KUKA KRL program: MyProgram_186().src

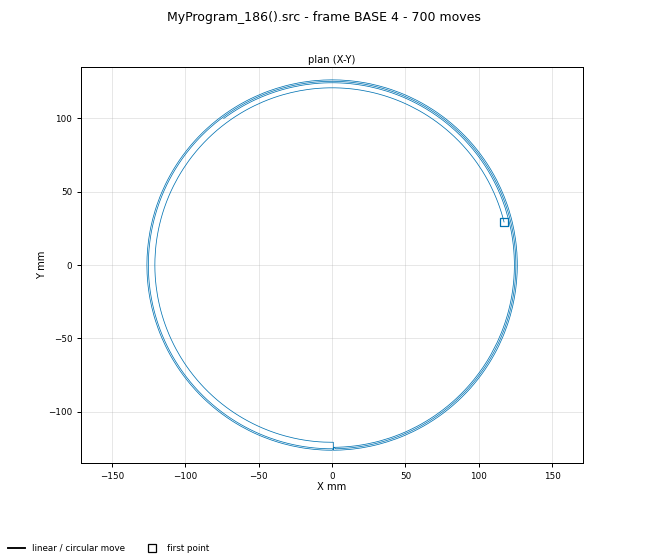
[picture p0: tool path of MyProgram_186().src in frame BASE 4, 700 of 700 moves have a stored position in this frame; points joined in program order, loops and branches not executed]
&ACCESS RVP
&REL 1
&PARAM TEMPLATE = C:\KRC\Roboter\Template\vorgabe
&PARAM EDITMASK = *
DEF MyProgram_186()
; ---- Setting reference (Base) ----
$BASE = BASE_DATA[4]

; --------------------------
; ---- Setting tool (TCP) ----
$TOOL = TOOL_DATA[3]
; --------------------------

$VEL.CP = VEL_APROX_PRINT
Startdeposition()
$VEL.CP = VEL_PRINT
LIN {X 117.2082,Y 29.362,Z 135,A 10.4187,B 24.9465,C -1.689,E1 25.1548,E2 795.6476} C_DIS
LIN {X 116.4539,Y 32.2231,Z 135,A 11.8113,B 24.9463,C -1.6929,E1 25.1537,E2 794.2539} C_DIS
LIN {X 115.5108,Y 35.4542,Z 135,A 13.5303,B 24.9456,C -1.7039,E1 25.1524,E2 792.5186} C_DIS
LIN {X 114.2566,Y 39.3095,Z 135,A 15.3056,B 24.9456,C -1.7024,E1 25.1508,E2 790.7568} C_DIS
LIN {X 113.2587,Y 42.0983,Z 135,A 16.7003,B 24.9454,C -1.7062,E1 25.1495,E2 789.3611} C_DIS
LIN {X 112.0398,Y 45.2414,Z 135,A 18.3803,B 24.9449,C -1.715,E1 25.1477,E2 787.6697} C_DIS
LIN {X 110.4582,Y 48.9779,Z 135,A 20.3068,B 24.9445,C -1.7207,E1 25.1456,E2 785.7402} C_DIS
LIN {X 109.0474,Y 52.0418,Z 135,A 21.6552,B 24.945,C -1.7129,E1 25.144,E2 784.4175} C_DIS
LIN {X 107.9261,Y 54.3318,Z 135,A 22.9862,B 24.9444,C -1.7224,E1 25.1423,E2 783.0713} C_DIS
LIN {X 106.3686,Y 57.3227,Z 135,A 24.664,B 24.9439,C -1.7307,E1 25.1401,E2 781.3826} C_DIS
LIN {X 104.398,Y 60.8384,Z 135,A 26.5827,B 24.9435,C -1.7363,E1 25.1375,E2 779.4606} C_DIS
LIN {X 102.3123,Y 64.2836,Z 135,A 28.5381,B 24.943,C -1.7437,E1 25.1346,E2 777.4977} C_DIS
LIN {X 100.337,Y 67.3254,Z 135,A 30.072,B 24.9433,C -1.7391,E1 25.1323,E2 775.9825} C_DIS
LIN {X 98.7776,Y 69.5926,Z 135,A 31.4665,B 24.9428,C -1.7468,E1 25.13,E2 774.5765} C_DIS
LIN {X 96.6464,Y 72.5239,Z 135,A 33.267,B 24.9423,C -1.7552,E1 25.127,E2 772.7648} C_DIS
LIN {X 93.8748,Y 76.0771,Z 135,A 35.2654,B 24.9423,C -1.7536,E1 25.1235,E2 770.7796} C_DIS
LIN {X 91.4934,Y 78.9247,Z 135,A 37.0151,B 24.9421,C -1.7572,E1 25.1204,E2 769.0292} C_DIS
LIN {X 89.0347,Y 81.6882,Z 135,A 38.7667,B 24.9419,C -1.7612,E1 25.1171,E2 767.2762} C_DIS
LIN {X 86.494,Y 84.3743,Z 135,A 40.6268,B 24.9413,C -1.7703,E1 25.1135,E2 765.4026} C_DIS
LIN {X 83.3087,Y 87.5205,Z 135,A 42.6146,B 24.9414,C -1.7682,E1 25.1095,E2 763.4279} C_DIS
LIN {X 80.5908,Y 90.0292,Z 135,A 44.3671,B 24.9412,C -1.7718,E1 25.1059,E2 761.6741} C_DIS
LIN {X 77.7969,Y 92.4543,Z 135,A 46.1818,B 24.9407,C -1.7782,E1 25.102,E2 759.8513} C_DIS
LIN {X 74.6844,Y 94.9862,Z 135,A 48.0527,B 24.9407,C -1.7802,E1 25.098,E2 757.9827} C_DIS
LIN {X 71.4297,Y 97.4574,Z 135,A 50.0698,B 24.9401,C -1.7875,E1 25.0934,E2 755.9555} C_DIS
LIN {X 68.3629,Y 99.6326,Z 135,A 51.6748,B 24.9405,C -1.782,E1 25.0898,E2 754.3691} C_DIS
LIN {X 65.5078,Y 101.5331,Z 135,A 53.2968,B 24.9403,C -1.7844,E1 25.086,E2 752.7466} C_DIS
LIN {X 62.4895,Y 103.4176,Z 135,A 55.0467,B 24.9399,C -1.7901,E1 25.0818,E2 750.989} C_DIS
LIN {X 59.1591,Y 105.3581,Z 135,A 56.9288,B 24.9396,C -1.7953,E1 25.0772,E2 749.1} C_DIS
LIN {X 55.2858,Y 107.4404,Z 135,A 58.8717,B 24.9399,C -1.7914,E1 25.0725,E2 747.172} C_DIS
LIN {X 53.0031,Y 108.5846,Z 135,A 60.0919,B 24.9397,C -1.7933,E1 25.0694,E2 745.9503} C_DIS
LIN {X 50.3072,Y 109.8593,Z 135,A 61.5505,B 24.9395,C -1.7972,E1 25.0657,E2 744.4864} C_DIS
LIN {X 47.239,Y 111.2147,Z 135,A 63.2747,B 24.9389,C -1.8053,E1 25.0612,E2 742.7473} C_DIS
LIN {X 43.152,Y 112.863,Z 135,A 65.1714,B 24.9394,C -1.7982,E1 25.0564,E2 740.8714} C_DIS
LIN {X 39.8076,Y 114.0839,Z 135,A 66.8981,B 24.9392,C -1.8016,E1 25.0518,E2 739.1402} C_DIS
LIN {X 35.4612,Y 115.5086,Z 135,A 69.1462,B 24.9388,C -1.8071,E1 25.0458,E2 736.8832} C_DIS
LIN {X 31.8058,Y 116.5702,Z 135,A 70.8147,B 24.9391,C -1.8019,E1 25.0414,E2 735.2298} C_DIS
LIN {X 28.3253,Y 117.4624,Z 135,A 72.5894,B 24.9388,C -1.8063,E1 25.0365,E2 733.4474} C_DIS
LIN {X 24.6405,Y 118.2916,Z 135,A 74.319,B 24.939,C -1.8043,E1 25.0318,E2 731.7247} C_DIS
LIN {X 21.612,Y 118.8814,Z 135,A 75.7474,B 24.939,C -1.8033,E1 25.0279,E2 730.3004} C_DIS
LIN {X 19.201,Y 119.2961,Z 135,A 77.0669,B 24.9385,C -1.8111,E1 25.0242,E2 728.9637} C_DIS
LIN {X 15.8744,Y 119.7824,Z 135,A 78.5695,B 24.9388,C -1.8073,E1 25.0201,E2 727.4715} C_DIS
LIN {X 12.9267,Y 120.1361,Z 135,A 80.0207,B 24.9386,C -1.8095,E1 25.0161,E2 726.0159} C_DIS
LIN {X 8.8957,Y 120.5018,Z 135,A 81.8563,B 24.9389,C -1.8058,E1 25.011,E2 724.1902} C_DIS
LIN {X 5.5184,Y 120.7048,Z 135,A 83.4356,B 24.9389,C -1.8046,E1 25.0066,E2 722.6143} C_DIS
LIN {X 1.8998,Y 120.8148,Z 135,A 85.2142,B 24.9388,C -1.8073,E1 25.0016,E2 720.8297} C_DIS
LIN {X -2.1053,Y 120.8114,Z 135,A 87.1828,B 24.9386,C -1.81,E1 24.9961,E2 718.8546} C_DIS
LIN {X -5.7963,Y 120.6909,Z 135,A 88.8573,B 24.9389,C -1.8059,E1 24.9915,E2 717.1894} C_DIS
LIN {X -9.3354,Y 120.4697,Z 135,A 90.493,B 24.9391,C -1.8031,E1 24.9869,E2 715.5598} C_DIS
LIN {X -12.922,Y 120.1366,Z 135,A 92.2805,B 24.9389,C -1.8059,E1 24.9819,E2 713.7647} C_DIS
LIN {X -16.2593,Y 119.7319,Z 135,A 93.9246,B 24.9388,C -1.8072,E1 24.9774,E2 712.1165} C_DIS
LIN {X -19.179,Y 119.2997,Z 135,A 95.2259,B 24.9392,C -1.8017,E1 24.9738,E2 710.8269} C_DIS
LIN {X -22.0873,Y 118.7951,Z 135,A 96.6396,B 24.9392,C -1.8013,E1 24.9699,E2 709.4128} C_DIS
LIN {X -25.0174,Y 118.2122,Z 135,A 98.0448,B 24.9393,C -1.7996,E1 24.9661,E2 708.0101} C_DIS
LIN {X -27.9199,Y 117.5601,Z 135,A 99.4567,B 24.9393,C -1.7983,E1 24.9622,E2 706.5992} C_DIS
LIN {X -30.7913,Y 116.8407,Z 135,A 100.8619,B 24.9395,C -1.797,E1 24.9585,E2 705.1951} C_DIS
LIN {X -33.6441,Y 116.0513,Z 135,A 102.2678,B 24.9395,C -1.7956,E1 24.9547,E2 703.7903} C_DIS
LIN {X -36.4781,Y 115.1919,Z 135,A 103.7338,B 24.9395,C -1.7967,E1 24.9508,E2 702.319} C_DIS
LIN {X -39.6947,Y 114.123,Z 135,A 105.3775,B 24.9395,C -1.7964,E1 24.9464,E2 700.6731} C_DIS
LIN {X -43.4807,Y 112.7353,Z 135,A 107.3067,B 24.9396,C -1.7946,E1 24.9414,E2 698.7442} C_DIS
LIN {X -47.2346,Y 111.2165,Z 135,A 109.2588,B 24.9397,C -1.7932,E1 24.9363,E2 696.7908} C_DIS
LIN {X -50.686,Y 109.6842,Z 135,A 110.9257,B 24.9403,C -1.785,E1 24.9321,E2 695.1394} C_DIS
LIN {X -52.9887,Y 108.5917,Z 135,A 112.1318,B 24.9404,C -1.7829,E1 24.9291,E2 693.9351} C_DIS
LIN {X -55.6297,Y 107.2632,Z 135,A 113.6217,B 24.9404,C -1.7845,E1 24.9254,E2 692.4374} C_DIS
LIN {X -59.1335,Y 105.3725,Z 135,A 115.5345,B 24.9404,C -1.7823,E1 24.9207,E2 690.5244} C_DIS
LIN {X -62.4785,Y 103.4242,Z 135,A 117.42,B 24.9405,C -1.7811,E1 24.9162,E2 688.636} C_DIS
LIN {X -66.2361,Y 101.0593,Z 135,A 119.3922,B 24.9412,C -1.7712,E1 24.9116,E2 686.6811} C_DIS
LIN {X -69.2054,Y 99.0495,Z 135,A 121.2054,B 24.9412,C -1.7727,E1 24.9074,E2 684.8581} C_DIS
LIN {X -72.4209,Y 96.7236,Z 135,A 123.1594,B 24.9412,C -1.7719,E1 24.903,E2 682.899} C_DIS
LIN {X -75.5035,Y 94.3369,Z 135,A 124.8973,B 24.9417,C -1.763,E1 24.8992,E2 681.1759} C_DIS
LIN {X -78.5173,Y 91.8438,Z 135,A 126.8819,B 24.9417,C -1.7645,E1 24.8949,E2 679.18} C_DIS
LIN {X -81.6855,Y 89.0372,Z 135,A 128.7832,B 24.9423,C -1.7552,E1 24.891,E2 677.2933} C_DIS
LIN {X -84.3863,Y 86.4823,Z 135,A 130.6628,B 24.9423,C -1.7561,E1 24.8872,E2 675.4039} C_DIS
LIN {X -87.5073,Y 83.3226,Z 135,A 132.6896,B 24.9428,C -1.7474,E1 24.8833,E2 673.389} C_DIS
LIN {X -90.2106,Y 80.3883,Z 135,A 134.6788,B 24.9428,C -1.7468,E1 24.8795,E2 671.3925} C_DIS
LIN {X -92.931,Y 77.2269,Z 135,A 136.6676,B 24.9431,C -1.7421,E1 24.876,E2 669.4058} C_DIS
LIN {X -95.7064,Y 73.76,Z 135,A 138.7691,B 24.9435,C -1.7362,E1 24.8723,E2 667.3083} C_DIS
LIN {X -97.9305,Y 70.7798,Z 135,A 140.4093,B 24.9442,C -1.726,E1 24.8697,E2 665.6845} C_DIS
LIN {X -99.6354,Y 68.3587,Z 135,A 141.8189,B 24.9444,C -1.7223,E1 24.8674,E2 664.2768} C_DIS
LIN {X -101.2806,Y 65.8967,Z 135,A 143.3404,B 24.9444,C -1.7234,E1 24.8651,E2 662.7451} C_DIS
LIN {X -103.4337,Y 62.4628,Z 135,A 145.2949,B 24.9446,C -1.7192,E1 24.8622,E2 660.7904} C_DIS
LIN {X -105.1225,Y 59.5778,Z 135,A 146.7644,B 24.9452,C -1.7096,E1 24.8602,E2 659.3363} C_DIS
LIN {X -106.7231,Y 56.6584,Z 135,A 148.3292,B 24.9456,C -1.7043,E1 24.8581,E2 657.7758} C_DIS
LIN {X -108.0429,Y 54.1013,Z 135,A 149.9082,B 24.9452,C -1.7094,E1 24.8561,E2 656.1762} C_DIS
LIN {X -109.854,Y 50.3187,Z 135,A 151.7779,B 24.946,C -1.6982,E1 24.8539,E2 654.3229} C_DIS
LIN {X -111.2154,Y 47.2373,Z 135,A 153.5277,B 24.9459,C -1.6998,E1 24.852,E2 652.5596} C_DIS
LIN {X -112.8752,Y 43.1207,Z 135,A 155.6091,B 24.9463,C -1.6923,E1 24.8498,E2 650.4845} C_DIS
LIN {X -114.3965,Y 38.9059,Z 135,A 157.5918,B 24.9471,C -1.6795,E1 24.848,E2 648.5212} C_DIS
LIN {X -115.5081,Y 35.4629,Z 135,A 159.3187,B 24.9475,C -1.6745,E1 24.8466,E2 646.7962} C_DIS
LIN {X -116.564,Y 31.829,Z 135,A 161.2881,B 24.9473,C -1.6762,E1 24.8451,E2 644.8112} C_DIS
LIN {X -117.6566,Y 27.5146,Z 135,A 163.257,B 24.9482,C -1.6634,E1 24.8438,E2 642.8615} C_DIS
LIN {X -118.3874,Y 24.1699,Z 135,A 164.9832,B 24.9482,C -1.6625,E1 24.8428,E2 641.1271} C_DIS
LIN {X -119.1212,Y 20.2495,Z 135,A 166.6304,B 24.9492,C -1.6459,E1 24.842,E2 639.5098} C_DIS
LIN {X -119.5811,Y 17.3261,Z 135,A 168.207,B 24.9491,C -1.6487,E1 24.8413,E2 637.917} C_DIS
LIN {X -120.0472,Y 13.7395,Z 135,A 170.0456,B 24.9491,C -1.6484,E1 24.8407,E2 636.0682} C_DIS
LIN {X -120.385,Y 10.3581,Z 135,A 171.5564,B 24.9497,C -1.6388,E1 24.8403,E2 634.5712} C_DIS
LIN {X -120.635,Y 6.878,Z 135,A 173.1938,B 24.9501,C -1.6326,E1 24.84,E2 632.9387} C_DIS
LIN {X -120.7635,Y 4.0528,Z 135,A 174.764,B 24.9497,C -1.6381,E1 24.8398,E2 631.3461} C_DIS
LIN {X -120.833,Y -0.0274,Z 135,A 176.6942,B 24.9501,C -1.6315,E1 24.8398,E2 629.4199} C_DIS
LIN {X -120.764,Y -4.0401,Z 135,A 178.5716,B 24.9506,C -1.6242,E1 24.8399,E2 627.5486} C_DIS
LIN {X -120.5782,Y -7.8,Z 135,A -179.7807,B 24.9513,C -1.6125,E1 24.8402,E2 625.9189} C_DIS
LIN {X -120.3476,Y -10.8007,Z 135,A -178.1521,B 24.951,C -1.6165,E1 24.8406,E2 624.2709} C_DIS
LIN {X -119.9212,Y -14.7964,Z 135,A -176.423,B 24.9519,C -1.6028,E1 24.8411,E2 622.5642} C_DIS
LIN {X -119.4614,Y -18.1345,Z 135,A -174.8931,B 24.9523,C -1.5948,E1 24.8417,E2 621.0444} C_DIS
LIN {X -119.0535,Y -20.6507,Z 135,A -173.5752,B 24.9523,C -1.5956,E1 24.8423,E2 619.7167} C_DIS
LIN {X -118.5115,Y -23.5602,Z 135,A -172.027,B 24.9522,C -1.5974,E1 24.8432,E2 618.155} C_DIS
LIN {X -117.6551,Y -27.5214,Z 135,A -170.1188,B 24.9526,C -1.5907,E1 24.8443,E2 616.2514} C_DIS
LIN {X -116.8402,Y -30.7932,Z 135,A -168.6255,B 24.9532,C -1.5812,E1 24.8454,E2 614.7721} C_DIS
LIN {X -116.0502,Y -33.648,Z 135,A -167.1399,B 24.9532,C -1.5804,E1 24.8465,E2 613.2798} C_DIS
LIN {X -114.8606,Y -37.5134,Z 135,A -165.1436,B 24.9534,C -1.5779,E1 24.8482,E2 611.2781} C_DIS
LIN {X -113.7612,Y -40.7209,Z 135,A -163.6662,B 24.954,C -1.5674,E1 24.8496,E2 609.8173} C_DIS
LIN {X -112.7305,Y -43.4928,Z 135,A -162.1512,B 24.954,C -1.5681,E1 24.8511,E2 608.292} C_DIS
LIN {X -111.2209,Y -47.224,Z 135,A -160.2057,B 24.9542,C -1.5641,E1 24.8532,E2 606.3453} C_DIS
LIN {X -109.689,Y -50.6756,Z 135,A -158.4301,B 24.9545,C -1.5583,E1 24.8552,E2 604.5738} C_DIS
LIN {X -107.9279,Y -54.3283,Z 135,A -156.6032,B 24.9551,C -1.5486,E1 24.8574,E2 602.7601} C_DIS
LIN {X -106.2929,Y -57.4635,Z 135,A -154.9304,B 24.9553,C -1.5438,E1 24.8596,E2 601.09} C_DIS
LIN {X -104.901,Y -59.9661,Z 135,A -153.6675,B 24.9558,C -1.5359,E1 24.8613,E2 599.8393} C_DIS
LIN {X -103.4277,Y -62.4727,Z 135,A -152.022,B 24.9553,C -1.5438,E1 24.8637,E2 598.1663} C_DIS
LIN {X -101.069,Y -66.2213,Z 135,A -150.0449,B 24.956,C -1.5329,E1 24.8667,E2 596.2053} C_DIS
LIN {X -99.0773,Y -69.1655,Z 135,A -148.2409,B 24.956,C -1.5338,E1 24.8695,E2 594.3903} C_DIS
LIN {X -96.8094,Y -72.3056,Z 135,A -146.4333,B 24.9563,C -1.5279,E1 24.8725,E2 592.5879} C_DIS
LIN {X -94.3688,Y -75.4635,Z 135,A -144.5488,B 24.9565,C -1.5229,E1 24.8758,E2 590.7064} C_DIS
LIN {X -91.978,Y -78.3594,Z 135,A -142.6987,B 24.9566,C -1.5218,E1 24.8791,E2 588.8505} C_DIS
LIN {X -89.3973,Y -81.2913,Z 135,A -140.8374,B 24.9568,C -1.5179,E1 24.8826,E2 586.99} C_DIS
LIN {X -87.3788,Y -83.457,Z 135,A -139.376,B 24.9568,C -1.5174,E1 24.8854,E2 585.5236} C_DIS
LIN {X -84.3803,Y -86.4881,Z 135,A -137.3443,B 24.9571,C -1.5135,E1 24.8894,E2 583.4926} C_DIS
LIN {X -81.2968,Y -89.3923,Z 135,A -135.4044,B 24.9575,C -1.5063,E1 24.8934,E2 581.562} C_DIS
LIN {X -78.3646,Y -91.9736,Z 135,A -133.5268,B 24.9576,C -1.5037,E1 24.8973,E2 579.6831} C_DIS
LIN {X -75.4202,Y -94.4033,Z 135,A -131.6828,B 24.9577,C -1.5018,E1 24.9013,E2 577.8366} C_DIS
LIN {X -71.9827,Y -97.0499,Z 135,A -129.7435,B 24.9582,C -1.4928,E1 24.9056,E2 575.9117} C_DIS
LIN {X -69.5654,Y -98.7967,Z 135,A -128.3274,B 24.9584,C -1.4905,E1 24.9088,E2 574.4963} C_DIS
LIN {X -66.7147,Y -100.7442,Z 135,A -126.5538,B 24.9582,C -1.494,E1 24.913,E2 572.7086} C_DIS
LIN {X -63.4025,Y -102.8607,Z 135,A -124.7161,B 24.9584,C -1.4899,E1 24.9173,E2 570.8747} C_DIS
LIN {X -60.8427,Y -104.3955,Z 135,A -123.251,B 24.9584,C -1.4901,E1 24.9209,E2 569.4048} C_DIS
LIN {X -57.3258,Y -106.3669,Z 135,A -121.2837,B 24.9584,C -1.49,E1 24.9257,E2 567.4321} C_DIS
LIN {X -53.9695,Y -108.1078,Z 135,A -119.6272,B 24.9589,C -1.4815,E1 24.9298,E2 565.7913} C_DIS
LIN {X -50.6934,Y -109.6808,Z 135,A -117.8275,B 24.9589,C -1.483,E1 24.9344,E2 563.9836} C_DIS
LIN {X -47.257,Y -111.2072,Z 135,A -115.9699,B 24.9587,C -1.4844,E1 24.9391,E2 562.1182} C_DIS
LIN {X -43.1096,Y -112.8795,Z 135,A -113.8737,B 24.9589,C -1.4812,E1 24.9446,E2 560.0251} C_DIS
LIN {X -38.9084,Y -114.3956,Z 135,A -111.9177,B 24.9594,C -1.4719,E1 24.9497,E2 558.0873} C_DIS
LIN {X -35.4668,Y -115.5069,Z 135,A -110.1223,B 24.9593,C -1.4743,E1 24.9545,E2 556.283} C_DIS
LIN {X -31.8386,Y -116.5614,Z 135,A -108.402,B 24.9595,C -1.4698,E1 24.9591,E2 554.5708} C_DIS
LIN {X -28.3319,Y -117.4608,Z 135,A -106.9397,B 24.9602,C -1.4571,E1 24.963,E2 553.1365} C_DIS
LIN {X -26.0933,Y -117.9799,Z 135,A -105.533,B 24.9595,C -1.4712,E1 24.9669,E2 551.6946} C_DIS
LIN {X -22.6913,Y -118.6797,Z 135,A -103.8665,B 24.9595,C -1.4714,E1 24.9715,E2 550.0255} C_DIS
LIN {X -19.2195,Y -119.2931,Z 135,A -102.1249,B 24.9593,C -1.4741,E1 24.9763,E2 548.2759} C_DIS
LIN {X -15.9428,Y -119.7734,Z 135,A -100.806,B 24.96,C -1.4621,E1 24.9799,E2 546.9846} C_DIS
LIN {X -12.9172,Y -120.1371,Z 135,A -99.1935,B 24.9595,C -1.4697,E1 24.9844,E2 545.3529} C_DIS
LIN {X -8.8875,Y -120.5024,Z 135,A -97.3386,B 24.9597,C -1.4666,E1 24.9895,E2 543.5044} C_DIS
LIN {X -5.5225,Y -120.7046,Z 135,A -95.7626,B 24.9597,C -1.4657,E1 24.9939,E2 541.9304} C_DIS
LIN {X -1.9035,Y -120.8148,Z 135,A -93.9063,B 24.9594,C -1.4725,E1 24.9991,E2 540.0577} C_DIS
LIN {X 0.8485,Y -120.8246,Z 135,A -92.9219,B 24.9602,C -1.4577,E1 25.0018,E2 539.1083} C_DIS
Enddeposition()
LIN {X 0.8961,Y -126.2488,Z 136,A -92.9261,B 24.9648,C -1.37,E1 25.0012,E2 539.3203} C_DIS
Startdeposition()
$VEL.CP = VEL_PRINT
LIN {X 3.4149,Y -126.2057,Z 136,A -91.4311,B 24.9639,C -1.3878,E1 25.0055,E2 537.7835} C_DIS
LIN {X 5.8456,Y -126.1173,Z 136,A -90.3974,B 24.9641,C -1.3847,E1 25.0084,E2 536.7575} C_DIS
LIN {X 9.0865,Y -125.9244,Z 136,A -88.8289,B 24.9638,C -1.3901,E1 25.0128,E2 535.1768} C_DIS
LIN {X 11.8893,Y -125.6908,Z 136,A -87.682,B 24.9641,C -1.3843,E1 25.0159,E2 534.0443} C_DIS
LIN {X 14.2304,Y -125.4492,Z 136,A -86.3353,B 24.9633,C -1.3988,E1 25.0197,E2 532.6641} C_DIS
LIN {X 17.5242,Y -125.03,Z 136,A -85.133,B 24.9641,C -1.3846,E1 25.023,E2 531.4964} C_DIS
LIN {X 20.067,Y -124.6487,Z 136,A -83.7089,B 24.9634,C -1.3983,E1 25.027,E2 530.0412} C_DIS
LIN {X 23.5227,Y -124.041,Z 136,A -82.3768,B 24.964,C -1.3866,E1 25.0306,E2 528.7384} C_DIS
LIN {X 25.9284,Y -123.5626,Z 136,A -80.9491,B 24.9631,C -1.4034,E1 25.0346,E2 527.2727} C_DIS
LIN {X 28.9638,Y -122.8859,Z 136,A -79.7386,B 24.9636,C -1.3946,E1 25.0378,E2 526.0846} C_DIS
LIN {X 32.1573,Y -122.0881,Z 136,A -78.3424,B 24.9637,C -1.3912,E1 25.0416,E2 524.6985} C_DIS
LIN {X 35.2045,Y -121.2442,Z 136,A -76.8451,B 24.9635,C -1.396,E1 25.0456,E2 523.1925} C_DIS
LIN {X 37.7031,Y -120.4926,Z 136,A -75.4783,B 24.9629,C -1.4066,E1 25.0493,E2 521.8029} C_DIS
LIN {X 41.1279,Y -119.3649,Z 136,A -74.1306,B 24.9636,C -1.3941,E1 25.0528,E2 520.4875} C_DIS
LIN {X 43.6551,Y -118.4656,Z 136,A -72.7856,B 24.9632,C -1.4022,E1 25.0564,E2 519.1262} C_DIS
LIN {X 46.7763,Y -117.2672,Z 136,A -71.3592,B 24.9633,C -1.3997,E1 25.0601,E2 517.7088} C_DIS
LIN {X 49.841,Y -115.9972,Z 136,A -69.8683,B 24.9633,C -1.4012,E1 25.0639,E2 516.2179} C_DIS
LIN {X 52.7402,Y -114.708,Z 136,A -68.3768,B 24.963,C -1.4061,E1 25.0677,E2 514.7185} C_DIS
LIN {X 55.1403,Y -113.5763,Z 136,A -67.0778,B 24.9626,C -1.4128,E1 25.071,E2 513.4069} C_DIS
LIN {X 58.2813,Y -111.995,Z 136,A -65.4414,B 24.9624,C -1.4177,E1 25.0751,E2 511.7636} C_DIS
LIN {X 62.1642,Y -109.889,Z 136,A -63.3723,B 24.962,C -1.4245,E1 25.0802,E2 509.6843} C_DIS
LIN {X 65.6751,Y -107.8276,Z 136,A -61.5639,B 24.962,C -1.426,E1 25.0845,E2 507.878} C_DIS
LIN {X 69.0964,Y -105.6678,Z 136,A -59.6893,B 24.9616,C -1.4316,E1 25.0889,E2 505.9963} C_DIS
LIN {X 72.7108,Y -103.2134,Z 136,A -57.7646,B 24.9616,C -1.4327,E1 25.0933,E2 504.0756} C_DIS
LIN {X 75.7271,Y -101.0219,Z 136,A -56.0226,B 24.9612,C -1.4389,E1 25.0973,E2 502.3252} C_DIS
LIN {X 79.202,Y -98.3204,Z 136,A -54.0798,B 24.9612,C -1.4405,E1 25.1015,E2 500.3859} C_DIS
LIN {X 82.5424,Y -95.5335,Z 136,A -52.1393,B 24.961,C -1.4433,E1 25.1057,E2 498.4463} C_DIS
LIN {X 85.7422,Y -92.6731,Z 136,A -50.1556,B 24.9606,C -1.4498,E1 25.1098,E2 496.4552} C_DIS
LIN {X 88.8161,Y -89.7307,Z 136,A -48.2267,B 24.9604,C -1.4545,E1 25.1136,E2 494.5234} C_DIS
LIN {X 91.8181,Y -86.6562,Z 136,A -46.3169,B 24.9602,C -1.4573,E1 25.1173,E2 492.6152} C_DIS
LIN {X 94.3412,Y -83.903,Z 136,A -44.6498,B 24.9601,C -1.4602,E1 25.1204,E2 490.9486} C_DIS
LIN {X 96.9888,Y -80.8281,Z 136,A -42.8457,B 24.9599,C -1.4632,E1 25.1237,E2 489.1458} C_DIS
LIN {X 99.546,Y -77.657,Z 136,A -40.9182,B 24.9594,C -1.4723,E1 25.127,E2 487.2057} C_DIS
LIN {X 101.9883,Y -74.4204,Z 136,A -39.1012,B 24.9592,C -1.4762,E1 25.1301,E2 485.3882} C_DIS
LIN {X 104.4674,Y -70.8974,Z 136,A -37.1868,B 24.959,C -1.4796,E1 25.1331,E2 483.4752} C_DIS
LIN {X 106.8508,Y -67.2517,Z 136,A -35.2888,B 24.9589,C -1.4812,E1 25.136,E2 481.583} C_DIS
LIN {X 108.7747,Y -64.0933,Z 136,A -33.5535,B 24.9585,C -1.4892,E1 25.1385,E2 479.8379} C_DIS
LIN {X 110.9686,Y -60.2155,Z 136,A -31.5536,B 24.9582,C -1.494,E1 25.1412,E2 477.8369} C_DIS
LIN {X 112.2771,Y -57.7365,Z 136,A -30.4887,B 24.9586,C -1.487,E1 25.1425,E2 476.7942} C_DIS
LIN {X 113.734,Y -54.8101,Z 136,A -29.06,B 24.9585,C -1.4886,E1 25.1443,E2 475.3693} C_DIS
LIN {X 115.1101,Y -51.8571,Z 136,A -27.6022,B 24.9583,C -1.4921,E1 25.146,E2 473.9113} C_DIS
LIN {X 116.2047,Y -49.3604,Z 136,A -26.0909,B 24.9573,C -1.5103,E1 25.1477,E2 472.3652} C_DIS
LIN {X 117.4643,Y -46.2805,Z 136,A -24.8023,B 24.9577,C -1.5034,E1 25.149,E2 471.1} C_DIS
LIN {X 118.6502,Y -43.1469,Z 136,A -23.1818,B 24.9571,C -1.5135,E1 25.1506,E2 469.4648} C_DIS
LIN {X 119.5932,Y -40.463,Z 136,A -21.997,B 24.9571,C -1.512,E1 25.1517,E2 468.2903} C_DIS
LIN {X 120.6039,Y -37.3403,Z 136,A -20.5857,B 24.9571,C -1.5127,E1 25.1529,E2 466.8854} C_DIS
LIN {X 121.5218,Y -34.2336,Z 136,A -18.9833,B 24.9565,C -1.5244,E1 25.1541,E2 465.2645} C_DIS
LIN {X 122.3556,Y -31.1214,Z 136,A -17.6048,B 24.9565,C -1.5247,E1 25.1551,E2 463.8932} C_DIS
LIN {X 123.0013,Y -28.4651,Z 136,A -16.4722,B 24.9565,C -1.523,E1 25.1558,E2 462.7712} C_DIS
LIN {X 123.5709,Y -25.8887,Z 136,A -14.9906,B 24.9555,C -1.5419,E1 25.1567,E2 461.2537} C_DIS
LIN {X 124.1542,Y -22.9276,Z 136,A -13.614,B 24.9552,C -1.5467,E1 25.1574,E2 459.8737} C_DIS
LIN {X 124.7195,Y -19.6111,Z 136,A -12.3467,B 24.9557,C -1.5381,E1 25.158,E2 458.6342} C_DIS
LIN {X 125.086,Y -17.1321,Z 136,A -10.9548,B 24.9547,C -1.5552,E1 25.1585,E2 457.2102} C_DIS
LIN {X 125.4891,Y -13.8597,Z 136,A -9.73,B 24.9552,C -1.5458,E1 25.1589,E2 456.0147} C_DIS
LIN {X 125.7447,Y -11.3251,Z 136,A -8.3294,B 24.9543,C -1.5625,E1 25.1593,E2 454.5831} C_DIS
LIN {X 126.0014,Y -7.949,Z 136,A -7.0916,B 24.9549,C -1.5519,E1 25.1595,E2 453.3778} C_DIS
LIN {X 126.1461,Y -5.171,Z 136,A -5.6647,B 24.9541,C -1.5647,E1 25.1597,E2 451.9292} C_DIS
LIN {X 126.2489,Y -0.8611,Z 136,A -3.715,B 24.9538,C -1.5708,E1 25.1597,E2 449.9767} C_DIS
LIN {X 126.2214,Y 2.8479,Z 136,A -1.9783,B 24.9533,C -1.5791,E1 25.1597,E2 448.2308} C_DIS
LIN {X 126.1141,Y 5.9103,Z 136,A -0.8401,B 24.9538,C -1.5704,E1 25.1596,E2 447.1198} C_DIS
LIN {X 125.9675,Y 8.4958,Z 136,A 0.6063,B 24.9527,C -1.5885,E1 25.1593,E2 445.6395} C_DIS
LIN {X 125.7097,Y 11.6919,Z 136,A 1.8047,B 24.9532,C -1.5797,E1 25.159,E2 444.4687} C_DIS
LIN {X 125.4492,Y 14.2304,Z 136,A 3.2144,B 24.9522,C -1.5967,E1 25.1586,E2 443.0274} C_DIS
LIN {X 125.039,Y 17.4608,Z 136,A 4.4117,B 24.9528,C -1.5867,E1 25.1582,E2 441.8606} C_DIS
LIN {X 124.5524,Y 20.6441,Z 136,A 5.9286,B 24.9524,C -1.5943,E1 25.1575,E2 440.3346} C_DIS
LIN {X 124.0497,Y 23.4772,Z 136,A 7.1658,B 24.9524,C -1.5949,E1 25.1569,E2 439.1033} C_DIS
LIN {X 123.5626,Y 25.9284,Z 136,A 8.5426,B 24.9514,C -1.6112,E1 25.1561,E2 437.6962} C_DIS
LIN {X 122.8721,Y 29.021,Z 136,A 9.7646,B 24.9518,C -1.6044,E1 25.1553,E2 436.4973} C_DIS
LIN {X 122.0769,Y 32.1989,Z 136,A 11.1361,B 24.9518,C -1.6031,E1 25.1544,E2 435.1369} C_DIS
LIN {X 121.2358,Y 35.2333,Z 136,A 12.6569,B 24.9513,C -1.6123,E1 25.1532,E2 433.603} C_DIS
LIN {X 120.4926,Y 37.7031,Z 136,A 14.0406,B 24.9504,C -1.627,E1 25.1521,E2 432.1925} C_DIS
LIN {X 119.4081,Y 41.0031,Z 136,A 15.3377,B 24.951,C -1.6173,E1 25.151,E2 430.9258} C_DIS
LIN {X 118.3423,Y 43.9842,Z 136,A 16.9118,B 24.9503,C -1.6288,E1 25.1494,E2 429.3333} C_DIS
LIN {X 117.3193,Y 46.647,Z 136,A 18.1017,B 24.9503,C -1.6272,E1 25.1482,E2 428.1538} C_DIS
LIN {X 116.0326,Y 49.7591,Z 136,A 19.5308,B 24.9504,C -1.6265,E1 25.1467,E2 426.7341} C_DIS
LIN {X 114.9165,Y 52.2895,Z 136,A 21.0882,B 24.9492,C -1.6459,E1 25.1449,E2 425.1395} C_DIS
LIN {X 113.505,Y 55.2848,Z 136,A 22.5502,B 24.9492,C -1.6481,E1 25.1431,E2 423.6801} C_DIS
LIN {X 112.1392,Y 58.0068,Z 136,A 23.9607,B 24.9488,C -1.6534,E1 25.1413,E2 422.2645} C_DIS
LIN {X 110.2513,Y 61.5196,Z 136,A 25.7324,B 24.9486,C -1.6565,E1 25.1389,E2 420.4949} C_DIS
LIN {X 108.1775,Y 65.0965,Z 136,A 27.6165,B 24.9482,C -1.662,E1 25.1362,E2 418.6075} C_DIS
LIN {X 105.7481,Y 68.9728,Z 136,A 29.5704,B 24.9482,C -1.6612,E1 25.1333,E2 416.6653} C_DIS
LIN {X 103.7966,Y 71.8762,Z 136,A 31.2616,B 24.9477,C -1.6707,E1 25.1306,E2 414.9601} C_DIS
LIN {X 101.0853,Y 75.642,Z 136,A 33.2385,B 24.9477,C -1.6693,E1 25.1274,E2 412.9959} C_DIS
LIN {X 98.7333,Y 78.6867,Z 136,A 35.0312,B 24.9474,C -1.676,E1 25.1243,E2 411.1957} C_DIS
LIN {X 95.9956,Y 82.0049,Z 136,A 36.9185,B 24.9473,C -1.6773,E1 25.1209,E2 409.314} C_DIS
LIN {X 93.6083,Y 84.7193,Z 136,A 38.6442,B 24.9468,C -1.6855,E1 25.1177,E2 407.5767} C_DIS
LIN {X 90.5252,Y 88.0063,Z 136,A 40.5964,B 24.9468,C -1.6853,E1 25.1139,E2 405.6334} C_DIS
LIN {X 87.9431,Y 90.5864,Z 136,A 42.3289,B 24.9463,C -1.6928,E1 25.1105,E2 403.8905} C_DIS
LIN {X 84.65,Y 93.6712,Z 136,A 44.2818,B 24.9463,C -1.6922,E1 25.1065,E2 401.947} C_DIS
LIN {X 81.9325,Y 96.057,Z 136,A 46.0134,B 24.9458,C -1.7001,E1 25.1028,E2 400.2036} C_DIS
LIN {X 78.5114,Y 98.8728,Z 136,A 47.9392,B 24.9458,C -1.6996,E1 25.0986,E2 398.2862} C_DIS
LIN {X 75.5727,Y 101.1369,Z 136,A 49.6925,B 24.9454,C -1.7062,E1 25.0947,E2 396.5236} C_DIS
LIN {X 71.9107,Y 103.7726,Z 136,A 51.6354,B 24.9456,C -1.7044,E1 25.0903,E2 394.5917} C_DIS
LIN {X 68.8956,Y 105.7983,Z 136,A 53.3637,B 24.9451,C -1.7112,E1 25.0862,E2 392.8532} C_DIS
LIN {X 65.1283,Y 108.1583,Z 136,A 55.3758,B 24.9449,C -1.714,E1 25.0815,E2 390.8406} C_DIS
LIN {X 61.4647,Y 110.2818,Z 136,A 57.3279,B 24.9447,C -1.7183,E1 25.0767,E2 388.8842} C_DIS
LIN {X 57.7288,Y 112.281,Z 136,A 58.988,B 24.9453,C -1.7078,E1 25.0727,E2 387.2537} C_DIS
LIN {X 54.7033,Y 113.785,Z 136,A 60.4271,B 24.9455,C -1.705,E1 25.0691,E2 385.825} C_DIS
LIN {X 52.2505,Y 114.9342,Z 136,A 61.9467,B 24.9445,C -1.721,E1 25.0652,E2 384.2715} C_DIS
LIN {X 49.3604,Y 116.2047,Z 136,A 63.4299,B 24.9442,C -1.7251,E1 25.0613,E2 382.7821} C_DIS
LIN {X 46.4345,Y 117.4044,Z 136,A 64.6895,B 24.9447,C -1.7178,E1 25.0581,E2 381.5425} C_DIS
LIN {X 43.1616,Y 118.6449,Z 136,A 66.3452,B 24.9444,C -1.7227,E1 25.0538,E2 379.8788} C_DIS
LIN {X 40.432,Y 119.6035,Z 136,A 67.5414,B 24.9447,C -1.718,E1 25.0506,E2 378.696} C_DIS
LIN {X 37.2586,Y 120.6289,Z 136,A 68.9391,B 24.945,C -1.7135,E1 25.047,E2 377.3116} C_DIS
LIN {X 34.2148,Y 121.5271,Z 136,A 70.4755,B 24.9446,C -1.7193,E1 25.0428,E2 375.764} C_DIS
LIN {X 31.5242,Y 122.2534,Z 136,A 71.8824,B 24.9441,C -1.7272,E1 25.039,E2 374.3407} C_DIS
LIN {X 28.6752,Y 122.9533,Z 136,A 73.1125,B 24.9444,C -1.7229,E1 25.0357,E2 373.1225} C_DIS
LIN {X 25.8887,Y 123.5709,Z 136,A 74.5669,B 24.9438,C -1.7314,E1 25.0316,E2 371.6499} C_DIS
LIN {X 22.7779,Y 124.181,Z 136,A 75.9747,B 24.9438,C -1.7305,E1 25.0278,E2 370.2459} C_DIS
LIN {X 19.4727,Y 124.741,Z 136,A 77.2967,B 24.9445,C -1.7212,E1 25.0242,E2 368.9471} C_DIS
LIN {X 17.1321,Y 125.086,Z 136,A 78.6191,B 24.9437,C -1.7336,E1 25.0205,E2 367.5965} C_DIS
LIN {X 13.7327,Y 125.5028,Z 136,A 79.865,B 24.9446,C -1.7189,E1 25.0171,E2 366.3864} C_DIS
LIN {X 11.3251,Y 125.7447,Z 136,A 81.2615,B 24.9437,C -1.7335,E1 25.0131,E2 364.9561} C_DIS
LIN {X 7.9619,Y 126.0006,Z 136,A 82.5568,B 24.9444,C -1.7221,E1 25.0096,E2 363.6884} C_DIS
LIN {X 5.6284,Y 126.1283,Z 136,A 83.8468,B 24.9437,C -1.7332,E1 25.0059,E2 362.3725} C_DIS
LIN {X 2.2947,Y 126.2311,Z 136,A 85.2055,B 24.9442,C -1.7255,E1 25.0022,E2 361.0323} C_DIS
LIN {X -0.1947,Y 126.2527,Z 136,A 86.2681,B 24.9444,C -1.7221,E1 24.9992,E2 359.9779} C_DIS
LIN {X -3.2029,Y 126.2115,Z 136,A 87.7454,B 24.9441,C -1.7271,E1 24.9951,E2 358.4885} C_DIS
LIN {X -5.9057,Y 126.1143,Z 136,A 88.9279,B 24.9443,C -1.7245,E1 24.9918,E2 357.3119} C_DIS
LIN {X -9.1355,Y 125.9208,Z 136,A 90.3717,B 24.9443,C -1.7228,E1 24.9878,E2 355.8718} C_DIS
LIN {X -11.829,Y 125.6966,Z 136,A 91.4898,B 24.9448,C -1.717,E1 24.9847,E2 354.767} C_DIS
LIN {X -14.2304,Y 125.4492,Z 136,A 92.8993,B 24.9438,C -1.7314,E1 24.9807,E2 353.3223} C_DIS
LIN {X -17.6112,Y 125.0175,Z 136,A 94.1257,B 24.9449,C -1.7151,E1 24.9774,E2 352.1336} C_DIS
LIN {X -20.067,Y 124.6487,Z 136,A 95.5471,B 24.944,C -1.7284,E1 24.9734,E2 350.6794} C_DIS
LIN {X -23.1676,Y 124.1089,Z 136,A 96.7577,B 24.9448,C -1.7169,E1 24.9702,E2 349.495} C_DIS
LIN {X -26.4185,Y 123.4567,Z 136,A 98.1677,B 24.9451,C -1.7111,E1 24.9663,E2 348.0969} C_DIS
LIN {X -28.8695,Y 122.9087,Z 136,A 99.5955,B 24.9443,C -1.7237,E1 24.9624,E2 346.6374} C_DIS
LIN {X -31.8142,Y 122.1795,Z 136,A 100.9829,B 24.9443,C -1.7228,E1 24.9586,E2 345.25} C_DIS
LIN {X -35.2575,Y 121.2287,Z 136,A 102.4365,B 24.945,C -1.7132,E1 24.9548,E2 343.8171} C_DIS
LIN {X -37.9662,Y 120.4085,Z 136,A 103.6795,B 24.9452,C -1.7097,E1 24.9514,E2 342.5801} C_DIS
LIN {X -41.0523,Y 119.3911,Z 136,A 105.1474,B 24.9454,C -1.7076,E1 24.9476,E2 341.1145} C_DIS
LIN {X -43.5727,Y 118.4964,Z 136,A 106.6462,B 24.9446,C -1.7194,E1 24.9436,E2 339.5846} C_DIS
LIN {X -46.6935,Y 117.3005,Z 136,A 107.9155,B 24.9455,C -1.7057,E1 24.9403,E2 338.3452} C_DIS
LIN {X -49.7635,Y 116.0307,Z 136,A 109.3557,B 24.9458,C -1.7003,E1 24.9366,E2 336.9144} C_DIS
LIN {X -52.5431,Y 114.7992,Z 136,A 110.9768,B 24.9452,C -1.7096,E1 24.9324,E2 335.2674} C_DIS
LIN {X -55.5483,Y 113.375,Z 136,A 112.2777,B 24.946,C -1.6974,E1 24.9292,E2 333.9921} C_DIS
LIN {X -58.3492,Y 111.9594,Z 136,A 113.8972,B 24.9456,C -1.7042,E1 24.9252,E2 332.3522} C_DIS
LIN {X -62.1231,Y 109.9121,Z 136,A 115.8314,B 24.9458,C -1.7,E1 24.9204,E2 330.4223} C_DIS
LIN {X -65.2338,Y 108.0945,Z 136,A 117.5531,B 24.9458,C -1.7011,E1 24.9163,E2 328.6929} C_DIS
LIN {X -68.7478,Y 105.8943,Z 136,A 119.4188,B 24.9461,C -1.6967,E1 24.9119,E2 326.8316} C_DIS
LIN {X -72.1386,Y 103.6141,Z 136,A 121.305,B 24.9461,C -1.6944,E1 24.9076,E2 324.9443} C_DIS
LIN {X -75.7271,Y 101.0219,Z 136,A 123.2319,B 24.9467,C -1.6864,E1 24.9033,E2 323.0298} C_DIS
LIN {X -78.6715,Y 98.7454,Z 136,A 125.016,B 24.9467,C -1.6871,E1 24.8993,E2 321.2374} C_DIS
LIN {X -82.0746,Y 95.9363,Z 136,A 127.0557,B 24.9468,C -1.6843,E1 24.895,E2 319.1965} C_DIS
LIN {X -85.149,Y 93.2184,Z 136,A 128.9009,B 24.9472,C -1.6792,E1 24.8911,E2 317.3563} C_DIS
LIN {X -88.1261,Y 90.409,Z 136,A 130.8143,B 24.9472,C -1.6773,E1 24.8873,E2 315.4395} C_DIS
LIN {X -91.1829,Y 87.3243,Z 136,A 132.759,B 24.9477,C -1.6712,E1 24.8835,E2 313.5009} C_DIS
LIN {X -93.7819,Y 84.5278,Z 136,A 134.5039,B 24.9479,C -1.6673,E1 24.8802,E2 311.7575} C_DIS
LIN {X -96.4575,Y 81.4614,Z 136,A 136.2986,B 24.9484,C -1.66,E1 24.877,E2 309.9719} C_DIS
LIN {X -99.0363,Y 78.306,Z 136,A 138.2702,B 24.9484,C -1.6607,E1 24.8735,E2 307.9895} C_DIS
LIN {X -101.675,Y 74.8469,Z 136,A 140.2031,B 24.9488,C -1.6534,E1 24.8703,E2 306.0647} C_DIS
LIN {X -103.8737,Y 71.7654,Z 136,A 141.9526,B 24.949,C -1.65,E1 24.8675,E2 304.3147} C_DIS
LIN {X -106.1502,Y 68.3527,Z 136,A 143.7367,B 24.9495,C -1.6411,E1 24.8648,E2 302.5427} C_DIS
LIN {X -108.2499,Y 64.9767,Z 136,A 145.6581,B 24.9495,C -1.6413,E1 24.862,E2 300.6112} C_DIS
LIN {X -110.4263,Y 61.2037,Z 136,A 147.6084,B 24.95,C -1.6342,E1 24.8593,E2 298.6675} C_DIS
LIN {X -112.1492,Y 57.9877,Z 136,A 149.3165,B 24.9501,C -1.6316,E1 24.8571,E2 296.9564} C_DIS
LIN {X -113.7034,Y 54.8742,Z 136,A 150.8209,B 24.9506,C -1.6235,E1 24.8552,E2 295.4634} C_DIS
LIN {X -115.1814,Y 51.6979,Z 136,A 152.2892,B 24.9512,C -1.6131,E1 24.8536,E2 294.0119} C_DIS
LIN {X -116.2047,Y 49.3604,Z 136,A 153.6639,B 24.9509,C -1.6193,E1 24.852,E2 292.6146} C_DIS
LIN {X -117.474,Y 46.2554,Z 136,A 154.9588,B 24.9518,C -1.6042,E1 24.8507,E2 291.3485} C_DIS
LIN {X -118.6607,Y 43.1179,Z 136,A 156.4546,B 24.9521,C -1.5983,E1 24.8492,E2 289.8584} C_DIS
LIN {X -119.5402,Y 40.622,Z 136,A 157.9141,B 24.9517,C -1.6061,E1 24.8479,E2 288.3718} C_DIS
LIN {X -120.505,Y 37.6634,Z 136,A 159.364,B 24.9518,C -1.6034,E1 24.8467,E2 286.9202} C_DIS
LIN {X -121.5337,Y 34.1911,Z 136,A 160.8702,B 24.9525,C -1.5919,E1 24.8455,E2 285.4327} C_DIS
LIN {X -122.2687,Y 31.4641,Z 136,A 162.0147,B 24.9531,C -1.5815,E1 24.8447,E2 284.3063} C_DIS
LIN {X -123.0239,Y 28.366,Z 136,A 163.4918,B 24.9533,C -1.5782,E1 24.8438,E2 282.8284} C_DIS
LIN {X -123.5709,Y 25.8887,Z 136,A 164.9243,B 24.9528,C -1.5872,E1 24.8429,E2 281.3661} C_DIS
LIN {X -124.1625,Y 22.8812,Z 136,A 166.3002,B 24.9531,C -1.5819,E1 24.8422,E2 279.9944} C_DIS
LIN {X -124.7075,Y 19.6888,Z 136,A 167.653,B 24.9537,C -1.5718,E1 24.8416,E2 278.6577} C_DIS
LIN {X -125.086,Y 17.1321,Z 136,A 168.8297,B 24.9539,C -1.5681,E1 24.8411,E2 277.4828} C_DIS
LIN {X -125.5056,Y 13.7062,Z 136,A 170.346,B 24.9544,C -1.5608,E1 24.8407,E2 275.975} C_DIS
LIN {X -125.7447,Y 11.3251,Z 136,A 171.4801,B 24.9544,C -1.5594,E1 24.8404,E2 274.8375} C_DIS
LIN {X -126.0007,Y 7.961,Z 136,A 172.8947,B 24.955,C -1.5491,E1 24.8401,E2 273.4389} C_DIS
LIN {X -126.1299,Y 5.5856,Z 136,A 174.0914,B 24.955,C -1.5508,E1 24.8399,E2 272.2308} C_DIS
LIN {X -126.223,Y 2.7834,Z 136,A 175.396,B 24.955,C -1.5481,E1 24.8399,E2 270.9249} C_DIS
LIN {X -126.2526,Y -0.1493,Z 136,A 176.6554,B 24.9555,C -1.5405,E1 24.8398,E2 269.676} C_DIS
LIN {X -126.2063,Y -3.3926,Z 136,A 178.1816,B 24.9557,C -1.5381,E1 24.8398,E2 268.1463} C_DIS
LIN {X -126.1162,Y -5.8679,Z 136,A 179.4561,B 24.9555,C -1.5413,E1 24.84,E2 266.8566} C_DIS
LIN {X -125.8992,Y -9.4315,Z 136,A -178.8997,B 24.9557,C -1.5371,E1 24.8403,E2 265.2124} C_DIS
LIN {X -125.5519,Y -13.2761,Z 136,A -177.4119,B 24.9567,C -1.5194,E1 24.8407,E2 263.7578} C_DIS
LIN {X -125.2067,Y -16.2108,Z 136,A -175.9557,B 24.9567,C -1.5203,E1 24.8412,E2 262.2908} C_DIS
LIN {X -124.6487,Y -20.067,Z 136,A -174.1204,B 24.9568,C -1.5177,E1 24.842,E2 260.4509} C_DIS
LIN {X -124.146,Y -22.9735,Z 136,A -172.6125,B 24.9567,C -1.5211,E1 24.8427,E2 258.9259} C_DIS
LIN {X -123.5319,Y -26.0705,Z 136,A -171.2419,B 24.9571,C -1.5137,E1 24.8435,E2 257.5647} C_DIS
LIN {X -122.9087,Y -28.8695,Z 136,A -169.9746,B 24.9574,C -1.5081,E1 24.8443,E2 256.3035} C_DIS
LIN {X -122.0581,Y -32.2695,Z 136,A -168.5699,B 24.9581,C -1.4946,E1 24.8453,E2 254.9226} C_DIS
LIN {X -121.3803,Y -34.7398,Z 136,A -167.0701,B 24.9575,C -1.5064,E1 24.8464,E2 253.386} C_DIS
LIN {X -120.4795,Y -37.7441,Z 136,A -165.7988,B 24.9581,C -1.4951,E1 24.8475,E2 252.1345} C_DIS
LIN {X -119.39,Y -41.0555,Z 136,A -164.2333,B 24.9584,C -1.4895,E1 24.8488,E2 250.5732} C_DIS
LIN {X -118.4964,Y -43.5727,Z 136,A -162.85,B 24.9582,C -1.4937,E1 24.8502,E2 249.1721} C_DIS
LIN {X -117.3251,Y -46.6326,Z 136,A -161.5511,B 24.9589,C -1.4807,E1 24.8515,E2 247.897} C_DIS
LIN {X -116.064,Y -49.6866,Z 136,A -160.1071,B 24.9593,C -1.4737,E1 24.853,E2 246.4616} C_DIS
LIN {X -114.7215,Y -52.7111,Z 136,A -158.6031,B 24.9595,C -1.4695,E1 24.8547,E2 244.9595} C_DIS
LIN {X -113.5763,Y -55.1403,Z 136,A -157.089,B 24.959,C -1.4795,E1 24.8566,E2 243.4132} C_DIS
LIN {X -112.0807,Y -58.1182,Z 136,A -155.5934,B 24.9593,C -1.4745,E1 24.8585,E2 241.9215} C_DIS
LIN {X -110.2513,Y -61.5196,Z 136,A -153.8291,B 24.9595,C -1.4702,E1 24.8609,E2 240.1583} C_DIS
LIN {X -108.2018,Y -65.0564,Z 136,A -151.9326,B 24.9597,C -1.4671,E1 24.8636,E2 238.2593} C_DIS
LIN {X -105.7388,Y -68.9872,Z 136,A -149.939,B 24.9603,C -1.4563,E1 24.8666,E2 236.2812} C_DIS
LIN {X -103.7269,Y -71.9765,Z 136,A -148.1973,B 24.9603,C -1.4571,E1 24.8693,E2 234.5292} C_DIS
LIN {X -101.4953,Y -75.0913,Z 136,A -146.4253,B 24.9603,C -1.4542,E1 24.8722,E2 232.7553} C_DIS
LIN {X -98.8282,Y -78.5674,Z 136,A -144.4785,B 24.9608,C -1.4474,E1 24.8756,E2 230.8155} C_DIS
LIN {X -96.0554,Y -81.9344,Z 136,A -142.5466,B 24.9611,C -1.4405,E1 24.879,E2 228.8912} C_DIS
LIN {X -93.5156,Y -84.8215,Z 136,A -140.7203,B 24.9611,C -1.4403,E1 24.8824,E2 227.0573} C_DIS
LIN {X -90.4674,Y -88.066,Z 136,A -138.6705,B 24.9613,C -1.4372,E1 24.8864,E2 225.006} C_DIS
LIN {X -87.5249,Y -90.9913,Z 136,A -136.8681,B 24.9617,C -1.4294,E1 24.89,E2 223.2146} C_DIS
LIN {X -84.6028,Y -93.714,Z 136,A -134.9662,B 24.9617,C -1.4299,E1 24.8939,E2 221.3038} C_DIS
LIN {X -81.4614,Y -96.4575,Z 136,A -133.1734,B 24.9622,C -1.4214,E1 24.8977,E2 219.5241} C_DIS
LIN {X -78.3978,Y -98.9632,Z 136,A -131.3561,B 24.9622,C -1.419,E1 24.9016,E2 217.7057} C_DIS
LIN {X -75.4479,Y -101.2298,Z 136,A -129.5822,B 24.9622,C -1.4201,E1 24.9056,E2 215.923} C_DIS
LIN {X -71.8443,Y -103.8188,Z 136,A -127.5419,B 24.9623,C -1.4179,E1 24.9103,E2 213.8809} C_DIS
LIN {X -68.4094,Y -106.1139,Z 136,A -125.7747,B 24.9628,C -1.4097,E1 24.9144,E2 212.1272} C_DIS
LIN {X -65.6751,Y -107.8276,Z 136,A -124.3111,B 24.9628,C -1.4075,E1 24.9178,E2 210.6645} C_DIS
LIN {X -62.2963,Y -109.814,Z 136,A -122.513,B 24.963,C -1.4058,E1 24.9222,E2 208.8649} C_DIS
LIN {X -58.9627,Y -111.6372,Z 136,A -120.8861,B 24.9633,C -1.3988,E1 24.9262,E2 207.25} C_DIS
LIN {X -56.5477,Y -112.882,Z 136,A -119.4362,B 24.9629,C -1.4076,E1 24.9298,E2 205.7753} C_DIS
LIN {X -53.4043,Y -114.4009,Z 136,A -117.9341,B 24.9632,C -1.4018,E1 24.9336,E2 204.2833} C_DIS
LIN {X -50.6037,Y -115.6674,Z 136,A -116.6704,B 24.9636,C -1.3939,E1 24.9368,E2 203.0352} C_DIS
LIN {X -47.5033,Y -116.9741,Z 136,A -115.1771,B 24.9638,C -1.3907,E1 24.9406,E2 201.5462} C_DIS
LIN {X -44.525,Y -118.1398,Z 136,A -113.5652,B 24.9634,C -1.3971,E1 24.9449,E2 199.9158} C_DIS
LIN {X -41.6775,Y -119.1743,Z 136,A -112.3621,B 24.9639,C -1.3875,E1 24.948,E2 198.7329} C_DIS
LIN {X -38.6508,Y -120.1898,Z 136,A -110.8468,B 24.9639,C -1.3896,E1 24.952,E2 197.2099} C_DIS
LIN {X -36.1921,Y -120.955,Z 136,A -109.4547,B 24.9633,C -1.3995,E1 24.9558,E2 195.7919} C_DIS
LIN {X -33.0996,Y -121.8368,Z 136,A -108.1238,B 24.9637,C -1.3923,E1 24.9593,E2 194.4759} C_DIS
LIN {X -29.8262,Y -122.678,Z 136,A -106.6656,B 24.9639,C -1.3878,E1 24.9633,E2 193.0265} C_DIS
LIN {X -27.3434,Y -123.2571,Z 136,A -105.3027,B 24.9634,C -1.3972,E1 24.967,E2 191.6394} C_DIS
LIN {X -24.0484,Y -123.9405,Z 136,A -104.0361,B 24.9641,C -1.3839,E1 24.9704,E2 190.4031} C_DIS
LIN {X -21.4031,Y -124.4258,Z 136,A -102.5939,B 24.9636,C -1.3943,E1 24.9745,E2 188.9347} C_DIS
LIN {X -18.4872,Y -124.8924,Z 136,A -101.4137,B 24.964,C -1.3861,E1 24.9777,E2 187.773} C_DIS
LIN {X -15.1329,Y -125.3416,Z 136,A -99.8395,B 24.964,C -1.3877,E1 24.9821,E2 186.1938} C_DIS
LIN {X -12.6058,Y -125.622,Z 136,A -98.7511,B 24.9641,C -1.3843,E1 24.9851,E2 185.1127} C_DIS
LIN {X -9.3675,Y -125.9039,Z 136,A -97.2366,B 24.9641,C -1.3862,E1 24.9893,E2 183.5931} C_DIS
LIN {X -6.8043,Y -126.0691,Z 136,A -96.1502,B 24.9642,C -1.3823,E1 24.9923,E2 182.5155} C_DIS
LIN {X -3.5797,Y -126.2011,Z 136,A -94.5814,B 24.9639,C -1.3877,E1 24.9967,E2 180.9338} C_DIS
LIN {X 0.1147,Y -126.2531,Z 136,A -92.962,B 24.9641,C -1.3852,E1 25.0012,E2 179.3203} C_DIS
LIN {X 0.1147,Y -126.2531,Z 136,A -92.962,B 24.9641,C -1.3852,E1 25.0012,E2 179.3203} C_DIS
Enddeposition()
LIN {X 0.8835,Y -125.2578,Z 136,A -92.5956,B 24.9631,C -1.4034,E1 25.0024,E2 178.9108} C_DIS
Startdeposition()
$VEL.CP = VEL_PRINT
LIN {X -3.1896,Y -125.2219,Z 136,A -95.135,B 24.9648,C -1.3699,E1 24.995,E2 181.5295} C_DIS
LIN {X -7.2132,Y -125.0552,Z 136,A -97.0396,B 24.965,C -1.3668,E1 24.9897,E2 183.4421} C_DIS
LIN {X -11.1339,Y -124.7677,Z 136,A -98.8407,B 24.965,C -1.3667,E1 24.9847,E2 185.2442} C_DIS
LIN {X -14.8551,Y -124.3781,Z 136,A -100.4554,B 24.9648,C -1.3716,E1 24.9802,E2 186.8483} C_DIS
LIN {X -18.8716,Y -123.8326,Z 136,A -102.3325,B 24.9648,C -1.3709,E1 24.975,E2 188.7285} C_DIS
LIN {X -22.5117,Y -123.2233,Z 136,A -104.113,B 24.965,C -1.3671,E1 24.9701,E2 190.5199} C_DIS
LIN {X -26.0701,Y -122.5195,Z 136,A -105.6998,B 24.9648,C -1.3713,E1 24.9658,E2 192.0986} C_DIS
LIN {X -29.9346,Y -121.6339,Z 136,A -107.6542,B 24.9651,C -1.3655,E1 24.9604,E2 194.0693} C_DIS
LIN {X -33.9009,Y -120.5873,Z 136,A -109.357,B 24.9646,C -1.375,E1 24.9559,E2 195.7523} C_DIS
LIN {X -37.6985,Y -119.4552,Z 136,A -111.25,B 24.9647,C -1.3725,E1 24.9508,E2 197.6544} C_DIS
LIN {X -42.5789,Y -117.8031,Z 136,A -113.523,B 24.9644,C -1.3785,E1 24.9449,E2 199.9175} C_DIS
LIN {X -45.7776,Y -116.598,Z 136,A -115.2244,B 24.9647,C -1.3735,E1 24.9404,E2 201.6345} C_DIS
LIN {X -49.4552,Y -115.0858,Z 136,A -116.8008,B 24.964,C -1.3868,E1 24.9364,E2 203.1828} C_DIS
LIN {X -52.2703,Y -113.835,Z 136,A -118.3911,B 24.9643,C -1.3799,E1 24.9323,E2 204.7934} C_DIS
LIN {X -55.4916,Y -112.2995,Z 136,A -119.9681,B 24.9641,C -1.3845,E1 24.9284,E2 206.3636} C_DIS
LIN {X -58.8471,Y -110.5802,Z 136,A -121.7697,B 24.9641,C -1.3831,E1 24.9239,E2 208.1733} C_DIS
LIN {X -61.9285,Y -108.8845,Z 136,A -123.3806,B 24.9641,C -1.3853,E1 24.92,E2 209.7838} C_DIS
LIN {X -65.3889,Y -106.8423,Z 136,A -125.2146,B 24.9639,C -1.3882,E1 24.9156,E2 211.6165} C_DIS
LIN {X -68.6093,Y -104.8037,Z 136,A -126.9283,B 24.9637,C -1.3924,E1 24.9115,E2 213.3258} C_DIS
LIN {X -71.6606,Y -102.7411,Z 136,A -128.6231,B 24.9636,C -1.3947,E1 24.9076,E2 215.0208} C_DIS
LIN {X -75.043,Y -100.2974,Z 136,A -130.6033,B 24.9636,C -1.3947,E1 24.9032,E2 217.0079} C_DIS
LIN {X -78.3854,Y -97.7076,Z 136,A -132.6259,B 24.9636,C -1.3943,E1 24.8987,E2 219.0391} C_DIS
LIN {X -82.0948,Y -94.6124,Z 136,A -134.7898,B 24.9632,C -1.4007,E1 24.8941,E2 221.1962} C_DIS
LIN {X -85.4226,Y -91.6184,Z 136,A -136.5833,B 24.9624,C -1.4166,E1 24.8905,E2 222.9591} C_DIS
LIN {X -88.03,Y -89.1168,Z 136,A -138.5137,B 24.9629,C -1.4073,E1 24.8866,E2 224.9195} C_DIS
LIN {X -91.2041,Y -85.8649,Z 136,A -140.5228,B 24.9625,C -1.4151,E1 24.8827,E2 226.9188} C_DIS
LIN {X -93.8259,Y -82.9919,Z 136,A -142.3509,B 24.9624,C -1.4169,E1 24.8793,E2 228.7507} C_DIS
LIN {X -96.5864,Y -79.7624,Z 136,A -144.2936,B 24.9621,C -1.4216,E1 24.8758,E2 230.6913} C_DIS
LIN {X -99.2628,Y -76.4068,Z 136,A -146.0558,B 24.9614,C -1.4355,E1 24.8728,E2 232.4287} C_DIS
LIN {X -101.3388,Y -73.6302,Z 136,A -147.8666,B 24.9617,C -1.4292,E1 24.8698,E2 234.2631} C_DIS
LIN {X -103.8652,Y -70.0215,Z 136,A -149.9916,B 24.9617,C -1.4295,E1 24.8664,E2 236.3981} C_DIS
LIN {X -106.5059,Y -65.9357,Z 136,A -152.1565,B 24.9613,C -1.4381,E1 24.8632,E2 238.5534} C_DIS
LIN {X -108.7361,Y -62.1887,Z 136,A -154.0866,B 24.9608,C -1.4464,E1 24.8605,E2 240.4736} C_DIS
LIN {X -110.6946,Y -58.6291,Z 136,A -155.9577,B 24.9606,C -1.451,E1 24.858,E2 242.3437} C_DIS
LIN {X -112.3433,Y -55.4027,Z 136,A -157.5379,B 24.9601,C -1.4592,E1 24.856,E2 243.9129} C_DIS
LIN {X -114.0047,Y -51.9034,Z 136,A -159.5011,B 24.9603,C -1.4557,E1 24.8537,E2 245.8952} C_DIS
LIN {X -115.6915,Y -48.0212,Z 136,A -161.3857,B 24.9599,C -1.4637,E1 24.8516,E2 247.7712} C_DIS
LIN {X -117.0449,Y -44.6266,Z 136,A -162.954,B 24.9593,C -1.4733,E1 24.85,E2 249.3255} C_DIS
LIN {X -118.1601,Y -41.5817,Z 136,A -164.5951,B 24.9595,C -1.4707,E1 24.8485,E2 250.982} C_DIS
LIN {X -119.3711,Y -37.9617,Z 136,A -166.3002,B 24.9591,C -1.4779,E1 24.847,E2 252.6797} C_DIS
LIN {X -120.5709,Y -33.9594,Z 136,A -168.1652,B 24.9586,C -1.4858,E1 24.8455,E2 254.5365} C_DIS
LIN {X -121.4354,Y -30.7244,Z 136,A -169.7233,B 24.9584,C -1.4894,E1 24.8444,E2 256.0951} C_DIS
LIN {X -122.249,Y -27.3146,Z 136,A -171.821,B 24.9594,C -1.4725,E1 24.8431,E2 258.2454} C_DIS
LIN {X -123.0543,Y -23.4136,Z 136,A -173.2868,B 24.9582,C -1.4941,E1 24.8424,E2 259.6685} C_DIS
LIN {X -123.762,Y -19.3275,Z 136,A -175.086,B 24.9576,C -1.5045,E1 24.8416,E2 261.4537} C_DIS
LIN {X -124.1683,Y -16.5187,Z 136,A -176.9573,B 24.9588,C -1.4834,E1 24.8409,E2 263.3865} C_DIS
LIN {X -124.6782,Y -12.0809,Z 136,A -178.4708,B 24.9571,C -1.5133,E1 24.8404,E2 264.8376} C_DIS
LIN {X -124.9228,Y -9.2148,Z 136,A -179.9027,B 24.9571,C -1.5125,E1 24.8401,E2 266.2802} C_DIS
LIN {X -125.1505,Y -5.3044,Z 136,A 178.3574,B 24.9567,C -1.5206,E1 24.8399,E2 268.0112} C_DIS
LIN {X -125.2567,Y -1.3589,Z 136,A 176.5323,B 24.9564,C -1.5256,E1 24.8398,E2 269.8353} C_DIS
LIN {X -125.2275,Y 2.9889,Z 136,A 174.4512,B 24.9563,C -1.5281,E1 24.8398,E2 271.9232} C_DIS
LIN {X -125.0193,Y 7.7962,Z 136,A 172.3493,B 24.9556,C -1.5397,E1 24.8402,E2 274.01} C_DIS
LIN {X -124.7966,Y 10.7921,Z 136,A 170.7171,B 24.956,C -1.5328,E1 24.8406,E2 275.6684} C_DIS
LIN {X -124.231,Y 16.0403,Z 136,A 168.8305,B 24.9542,C -1.5641,E1 24.8411,E2 277.4917} C_DIS
LIN {X -123.6328,Y 20.1425,Z 136,A 166.6134,B 24.9546,C -1.556,E1 24.8421,E2 279.7412} C_DIS
LIN {X -123.0353,Y 23.5132,Z 136,A 165.0354,B 24.9544,C -1.5606,E1 24.8429,E2 281.3177} C_DIS
LIN {X -122.4125,Y 26.566,Z 136,A 163.1187,B 24.9554,C -1.5436,E1 24.8441,E2 283.2862} C_DIS
LIN {X -121.431,Y 30.7417,Z 136,A 161.6617,B 24.9537,C -1.5722,E1 24.845,E2 284.6836} C_DIS
LIN {X -120.5,Y 34.2129,Z 136,A 159.821,B 24.9539,C -1.5687,E1 24.8464,E2 286.5432} C_DIS
LIN {X -119.3634,Y 37.9858,Z 136,A 158.2087,B 24.9531,C -1.5829,E1 24.8477,E2 288.1309} C_DIS
LIN {X -118.266,Y 41.2762,Z 136,A 156.5942,B 24.9528,C -1.5867,E1 24.8491,E2 289.7457} C_DIS
LIN {X -117.0603,Y 44.5855,Z 136,A 154.8617,B 24.9528,C -1.5863,E1 24.8508,E2 291.4888} C_DIS
LIN {X -115.7428,Y 47.8984,Z 136,A 153.3066,B 24.9523,C -1.5948,E1 24.8525,E2 293.0324} C_DIS
LIN {X -114.4059,Y 51.0079,Z 136,A 151.8216,B 24.9519,C -1.6024,E1 24.8541,E2 294.5074} C_DIS
LIN {X -112.717,Y 54.6433,Z 136,A 149.5784,B 24.9526,C -1.5898,E1 24.8569,E2 296.7929} C_DIS
LIN {X -111.18,Y 57.7047,Z 136,A 148.2764,B 24.9517,C -1.6062,E1 24.8585,E2 298.0627} C_DIS
LIN {X -108.9978,Y 61.7299,Z 136,A 146.1865,B 24.9513,C -1.6126,E1 24.8613,E2 300.1483} C_DIS
LIN {X -106.9676,Y 65.1844,Z 136,A 144.4449,B 24.9507,C -1.622,E1 24.8638,E2 301.8765} C_DIS
LIN {X -104.2204,Y 69.4914,Z 136,A 142.0151,B 24.9505,C -1.6246,E1 24.8675,E2 304.3125} C_DIS
LIN {X -102.065,Y 72.6207,Z 136,A 140.2517,B 24.9503,C -1.6283,E1 24.8703,E2 306.0757} C_DIS
LIN {X -99.7811,Y 75.7285,Z 136,A 138.3369,B 24.9504,C -1.6264,E1 24.8735,E2 308.0042} C_DIS
LIN {X -96.506,Y 79.8595,Z 136,A 135.7693,B 24.9504,C -1.6259,E1 24.8781,E2 310.585} C_DIS
LIN {X -94.3143,Y 82.4365,Z 136,A 134.5069,B 24.9494,C -1.6426,E1 24.8803,E2 311.8132} C_DIS
LIN {X -92.2496,Y 84.7406,Z 136,A 132.9882,B 24.9495,C -1.6416,E1 24.8832,E2 313.341} C_DIS
LIN {X -89.1928,Y 87.9528,Z 136,A 130.9772,B 24.9491,C -1.6474,E1 24.8871,E2 315.3469} C_DIS
LIN {X -85.5749,Y 91.4766,Z 136,A 128.6639,B 24.9488,C -1.6529,E1 24.8918,E2 317.6567} C_DIS
LIN {X -83.2937,Y 93.5588,Z 136,A 127.178,B 24.9488,C -1.6529,E1 24.8949,E2 319.1485} C_DIS
LIN {X -79.6671,Y 96.6653,Z 136,A 125.1162,B 24.9482,C -1.6633,E1 24.8992,E2 321.1934} C_DIS
LIN {X -75.7479,Y 99.7664,Z 136,A 122.7793,B 24.948,C -1.666,E1 24.9044,E2 323.5326} C_DIS
LIN {X -72.5544,Y 102.1124,Z 136,A 120.9373,B 24.9478,C -1.6684,E1 24.9085,E2 325.3752} C_DIS
LIN {X -70.0458,Y 103.8487,Z 136,A 119.0325,B 24.9491,C -1.6482,E1 24.9131,E2 327.3344} C_DIS
LIN {X -66.1425,Y 106.3773,Z 136,A 117.5095,B 24.9471,C -1.6796,E1 24.9165,E2 328.7876} C_DIS
LIN {X -63.1713,Y 108.1685,Z 136,A 115.7882,B 24.9473,C -1.6764,E1 24.9207,E2 330.5218} C_DIS
LIN {X -59.2841,Y 110.3465,Z 136,A 113.8552,B 24.9468,C -1.6848,E1 24.9254,E2 332.4403} C_DIS
LIN {X -55.8456,Y 112.1249,Z 136,A 112.043,B 24.9468,C -1.6858,E1 24.9299,E2 334.2549} C_DIS
LIN {X -53.0414,Y 113.4783,Z 136,A 110.1871,B 24.9478,C -1.6684,E1 24.9347,E2 336.157} C_DIS
LIN {X -49.4226,Y 115.1,Z 136,A 108.4882,B 24.9473,C -1.6763,E1 24.939,E2 337.8411} C_DIS
LIN {X -46.1507,Y 116.4523,Z 136,A 107.0894,B 24.9466,C -1.6886,E1 24.9426,E2 339.2136} C_DIS
LIN {X -42.9763,Y 117.6597,Z 136,A 105.5402,B 24.9464,C -1.6909,E1 24.9466,E2 340.7607} C_DIS
LIN {X -39.4137,Y 118.8996,Z 136,A 104.1375,B 24.9453,C -1.708,E1 24.9502,E2 342.1254} C_DIS
LIN {X -35.1232,Y 120.2368,Z 136,A 101.8966,B 24.9457,C -1.7017,E1 24.9563,E2 344.385} C_DIS
LIN {X -29.2426,Y 121.8008,Z 136,A 98.7471,B 24.9466,C -1.6875,E1 24.9649,E2 347.5728} C_DIS
LIN {X -25.9659,Y 122.5418,Z 136,A 97.3494,B 24.9461,C -1.6953,E1 24.9687,E2 348.9537} C_DIS
LIN {X -21.7183,Y 123.3653,Z 136,A 95.4298,B 24.9459,C -1.6996,E1 24.9739,E2 350.865} C_DIS
LIN {X -17.6905,Y 124.0065,Z 136,A 93.8353,B 24.945,C -1.7136,E1 24.9782,E2 352.4278} C_DIS
LIN {X -14.1847,Y 124.4581,Z 136,A 91.9991,B 24.9456,C -1.7043,E1 24.9834,E2 354.2874} C_DIS
LIN {X -10.8035,Y 124.7956,Z 136,A 90.471,B 24.9454,C -1.7063,E1 24.9876,E2 355.8116} C_DIS
LIN {X -7.0088,Y 125.0678,Z 136,A 88.6743,B 24.9456,C -1.7043,E1 24.9926,E2 357.6136} C_DIS
LIN {X -3.3985,Y 125.2161,Z 136,A 87.1246,B 24.9452,C -1.7097,E1 24.9969,E2 359.1508} C_DIS
LIN {X 0.527,Y 125.2612,Z 136,A 85.3705,B 24.9451,C -1.712,E1 25.0018,E2 360.8993} C_DIS
LIN {X 3.7596,Y 125.2061,Z 136,A 83.8426,B 24.9452,C -1.7099,E1 25.0061,E2 362.432} C_DIS
LIN {X 7.6966,Y 125.0255,Z 136,A 82.0361,B 24.9452,C -1.7098,E1 25.0111,E2 364.2381} C_DIS
LIN {X 11.5498,Y 124.7292,Z 136,A 80.2044,B 24.9454,C -1.7066,E1 25.0162,E2 366.0765} C_DIS
LIN {X 15.7189,Y 124.2731,Z 136,A 78.3208,B 24.9454,C -1.7078,E1 25.0215,E2 367.9556} C_DIS
LIN {X 19.3932,Y 123.7519,Z 136,A 76.6052,B 24.9454,C -1.7065,E1 25.0262,E2 369.6728} C_DIS
LIN {X 23.411,Y 123.0549,Z 136,A 74.7919,B 24.9454,C -1.7083,E1 25.0312,E2 371.4799} C_DIS
LIN {X 26.5644,Y 122.4128,Z 136,A 73.2821,B 24.9454,C -1.7057,E1 25.0353,E2 372.9938} C_DIS
LIN {X 30.4339,Y 121.5091,Z 136,A 71.4742,B 24.9455,C -1.7051,E1 25.0402,E2 374.8005} C_DIS
LIN {X 33.519,Y 120.6941,Z 136,A 70.0126,B 24.9455,C -1.7041,E1 25.0441,E2 376.2623} C_DIS
LIN {X 36.5253,Y 119.8184,Z 136,A 68.3759,B 24.9463,C -1.6931,E1 25.0486,E2 377.922} C_DIS
LIN {X 40.9044,Y 118.3949,Z 136,A 66.5572,B 24.9455,C -1.7052,E1 25.0533,E2 379.7085} C_DIS
LIN {X 43.9218,Y 117.3089,Z 136,A 65.0416,B 24.9457,C -1.7015,E1 25.0573,E2 381.2298} C_DIS
LIN {X 47.7207,Y 115.8171,Z 136,A 63.1793,B 24.9459,C -1.6998,E1 25.0621,E2 383.0921} C_DIS
LIN {X 50.8948,Y 114.4565,Z 136,A 61.6134,B 24.9459,C -1.6987,E1 25.0661,E2 384.6567} C_DIS
LIN {X 53.5662,Y 113.2315,Z 136,A 60.2363,B 24.9461,C -1.6954,E1 25.0696,E2 386.038} C_DIS
LIN {X 55.975,Y 112.061,Z 136,A 58.9374,B 24.9465,C -1.6902,E1 25.0729,E2 387.3457} C_DIS
LIN {X 59.5526,Y 110.2022,Z 136,A 57.3941,B 24.9457,C -1.7025,E1 25.0766,E2 388.8556} C_DIS
LIN {X 63.7319,Y 107.8392,Z 136,A 54.9135,B 24.9468,C -1.6852,E1 25.0827,E2 391.3696} C_DIS
LIN {X 67.3109,Y 105.6421,Z 136,A 53.0123,B 24.9469,C -1.6832,E1 25.0872,E2 393.2695} C_DIS
LIN {X 71.0207,Y 103.1845,Z 136,A 51.0041,B 24.947,C -1.6811,E1 25.0919,E2 395.2758} C_DIS
LIN {X 74.4733,Y 100.7215,Z 136,A 49.2947,B 24.9465,C -1.6892,E1 25.0957,E2 396.9603} C_DIS
LIN {X 77.1956,Y 98.6501,Z 136,A 47.4799,B 24.9475,C -1.6738,E1 25.0998,E2 398.8046} C_DIS
LIN {X 80.7319,Y 95.7778,Z 136,A 45.5503,B 24.9473,C -1.6775,E1 25.1039,E2 400.7183} C_DIS
LIN {X 83.3987,Y 93.4647,Z 136,A 43.802,B 24.9479,C -1.6676,E1 25.1076,E2 402.483} C_DIS
LIN {X 86.7266,Y 90.3853,Z 136,A 41.7586,B 24.9481,C -1.6647,E1 25.1117,E2 404.5247} C_DIS
LIN {X 89.6801,Y 87.4559,Z 136,A 39.9101,B 24.9481,C -1.6633,E1 25.1154,E2 406.3689} C_DIS
LIN {X 92.5237,Y 84.4419,Z 136,A 37.9685,B 24.9486,C -1.6567,E1 25.1191,E2 408.3176} C_DIS
LIN {X 95.083,Y 81.549,Z 136,A 36.2858,B 24.9486,C -1.6567,E1 25.1221,E2 409.9925} C_DIS
LIN {X 97.4623,Y 78.6895,Z 136,A 34.5383,B 24.949,C -1.6503,E1 25.1252,E2 411.747} C_DIS
LIN {X 100.1569,Y 75.2305,Z 136,A 32.5292,B 24.9493,C -1.6452,E1 25.1287,E2 413.7587} C_DIS
LIN {X 102.6107,Y 71.848,Z 136,A 30.6006,B 24.9496,C -1.6394,E1 25.1318,E2 415.6915} C_DIS
LIN {X 105.0556,Y 68.2222,Z 136,A 28.6911,B 24.9496,C -1.6388,E1 25.1347,E2 417.593} C_DIS
LIN {X 107.1081,Y 64.9526,Z 136,A 26.9227,B 24.95,C -1.6339,E1 25.1373,E2 419.364} C_DIS
LIN {X 109.0788,Y 61.586,Z 136,A 25.1007,B 24.9504,C -1.6271,E1 25.1399,E2 421.1927} C_DIS
LIN {X 110.7334,Y 58.5553,Z 136,A 23.72,B 24.95,C -1.6328,E1 25.1417,E2 422.5526} C_DIS
LIN {X 112.9204,Y 54.2173,Z 136,A 21.0721,B 24.9517,C -1.6048,E1 25.145,E2 425.2523} C_DIS
LIN {X 114.3402,Y 51.1547,Z 136,A 19.8544,B 24.951,C -1.6169,E1 25.1464,E2 426.4348} C_DIS
LIN {X 115.9291,Y 47.4489,Z 136,A 17.9488,B 24.9515,C -1.6083,E1 25.1484,E2 428.3502} C_DIS
LIN {X 117.2785,Y 44.003,Z 136,A 16.3904,B 24.9515,C -1.6102,E1 25.15,E2 429.8957} C_DIS
LIN {X 118.378,Y 40.9531,Z 136,A 15.072,B 24.9512,C -1.6141,E1 25.1512,E2 431.1973} C_DIS
LIN {X 119.8423,Y 36.4472,Z 136,A 12.7425,B 24.9521,C -1.5991,E1 25.1532,E2 433.549} C_DIS
LIN {X 120.8861,Y 32.824,Z 136,A 10.9773,B 24.9525,C -1.5917,E1 25.1545,E2 435.3216} C_DIS
LIN {X 121.789,Y 29.2915,Z 136,A 9.4517,B 24.9525,C -1.5937,E1 25.1556,E2 436.8335} C_DIS
LIN {X 122.4509,Y 26.3881,Z 136,A 7.7848,B 24.9536,C -1.5738,E1 25.1566,E2 438.5378} C_DIS
LIN {X 123.4615,Y 21.1691,Z 136,A 5.5682,B 24.9534,C -1.577,E1 25.1577,E2 440.7338} C_DIS
LIN {X 124.0222,Y 17.5807,Z 136,A 3.9816,B 24.9534,C -1.5755,E1 25.1583,E2 442.3145} C_DIS
LIN {X 124.506,Y 13.7463,Z 136,A 2.2738,B 24.9536,C -1.5729,E1 25.1589,E2 444.0184} C_DIS
LIN {X 124.819,Y 10.5268,Z 136,A 0.708,B 24.9542,C -1.5637,E1 25.1593,E2 445.5967} C_DIS
LIN {X 125.0952,Y 6.4675,Z 136,A -1.1407,B 24.9545,C -1.5582,E1 25.1596,E2 447.4473} C_DIS
LIN {X 125.236,Y 2.617,Z 136,A -2.9358,B 24.9549,C -1.5507,E1 25.1598,E2 449.2493} C_DIS
LIN {X 125.2573,Y -1.2346,Z 136,A -4.7561,B 24.9555,C -1.5419,E1 25.1598,E2 451.0796} C_DIS
LIN {X 125.1429,Y -5.4996,Z 136,A -6.6558,B 24.9557,C -1.5382,E1 25.1596,E2 452.9769} C_DIS
LIN {X 124.901,Y -9.5128,Z 136,A -8.5,B 24.956,C -1.5319,E1 25.1592,E2 454.8249} C_DIS
LIN {X 124.5652,Y -13.1961,Z 136,A -10.0652,B 24.956,C -1.5328,E1 25.1588,E2 456.3786} C_DIS
LIN {X 124.1614,Y -16.5718,Z 136,A -11.7338,B 24.9566,C -1.5219,E1 25.1582,E2 458.0632} C_DIS
LIN {X 123.5459,Y -20.6637,Z 136,A -13.4975,B 24.9566,C -1.5223,E1 25.1574,E2 459.8155} C_DIS
LIN {X 122.8904,Y -24.27,Z 136,A -15.229,B 24.9571,C -1.5139,E1 25.1565,E2 461.5565} C_DIS
LIN {X 122.2803,Y -27.1775,Z 136,A -16.4563,B 24.9569,C -1.5163,E1 25.1558,E2 462.7712} C_DIS
LIN {X 121.299,Y -31.262,Z 136,A -18.5283,B 24.9577,C -1.5023,E1 25.1544,E2 464.8642} C_DIS
LIN {X 120.3007,Y -34.9049,Z 136,A -20.1387,B 24.9577,C -1.5028,E1 25.1532,E2 466.4642} C_DIS
LIN {X 119.4534,Y -37.7042,Z 136,A -22.0725,B 24.9596,C -1.4679,E1 25.1515,E2 468.4692} C_DIS
LIN {X 117.9534,Y -42.1619,Z 136,A -23.616,B 24.9583,C -1.4923,E1 25.1501,E2 469.9466} C_DIS
LIN {X 116.9075,Y -44.9815,Z 136,A -25.026,B 24.9586,C -1.4861,E1 25.1487,E2 471.3633} C_DIS
LIN {X 114.7914,Y -50.1362,Z 136,A -27.6145,B 24.9592,C -1.4761,E1 25.1459,E2 473.9611} C_DIS
LIN {X 113.1324,Y -53.7736,Z 136,A -29.3182,B 24.9592,C -1.477,E1 25.1439,E2 475.6537} C_DIS
LIN {X 110.1768,Y -59.5999,Z 136,A -32.3725,B 24.9598,C -1.4645,E1 25.14,E2 478.7212} C_DIS
LIN {X 108.1699,Y -63.1691,Z 136,A -34.2551,B 24.9602,C -1.4584,E1 25.1374,E2 480.6083} C_DIS
LIN {X 106.2922,Y -66.2792,Z 136,A -35.9231,B 24.9604,C -1.4533,E1 25.1349,E2 482.28} C_DIS
LIN {X 103.8681,Y -70.0173,Z 136,A -37.8895,B 24.9606,C -1.4511,E1 25.1319,E2 484.2418} C_DIS
LIN {X 102.2264,Y -72.3931,Z 136,A -39.27,B 24.9609,C -1.4443,E1 25.1297,E2 485.6315} C_DIS
LIN {X 99.5132,Y -76.0793,Z 136,A -41.2303,B 24.9609,C -1.4453,E1 25.1264,E2 487.58} C_DIS
LIN {X 97.6157,Y -78.4994,Z 136,A -43.5993,B 24.9637,C -1.3927,E1 25.1221,E2 490.062} C_DIS
LIN {X 93.384,Y -83.4888,Z 136,A -45.48,B 24.9611,C -1.4412,E1 25.1188,E2 491.82} C_DIS
LIN {X 90.4446,Y -86.6637,Z 136,A -47.7076,B 24.962,C -1.4235,E1 25.1145,E2 494.0797} C_DIS
LIN {X 84.3993,Y -92.5624,Z 136,A -51.2524,B 24.9617,C -1.4302,E1 25.1074,E2 497.5939} C_DIS
LIN {X 79.6661,Y -96.6661,Z 136,A -54.8944,B 24.9641,C -1.3843,E1 25.0995,E2 501.33} C_DIS
LIN {X 75.859,Y -99.6817,Z 136,A -56.5668,B 24.9629,C -1.4071,E1 25.0959,E2 502.9425} C_DIS
LIN {X 72.3546,Y -102.2536,Z 136,A -58.5258,B 24.9631,C -1.4044,E1 25.0915,E2 504.9011} C_DIS
LIN {X 68.718,Y -104.7321,Z 136,A -60.5265,B 24.9632,C -1.4009,E1 25.0868,E2 506.9033} C_DIS
LIN {X 66.0496,Y -106.435,Z 136,A -62.0098,B 24.9635,C -1.3963,E1 25.0833,E2 508.3926} C_DIS
LIN {X 62.5846,Y -108.5088,Z 136,A -63.7955,B 24.9635,C -1.396,E1 25.079,E2 510.1738} C_DIS
LIN {X 59.5977,Y -110.178,Z 136,A -65.2326,B 24.9633,C -1.3996,E1 25.0755,E2 511.5981} C_DIS
LIN {X 56.8646,Y -111.6105,Z 136,A -66.9845,B 24.9643,C -1.3802,E1 25.0711,E2 513.391} C_DIS
LIN {X 52.5753,Y -113.694,Z 136,A -68.8006,B 24.9636,C -1.3949,E1 25.0666,E2 515.1676} C_DIS
LIN {X 50.0608,Y -114.824,Z 136,A -70.116,B 24.9638,C -1.3902,E1 25.0632,E2 516.491} C_DIS
LIN {X 47.2367,Y -116.0146,Z 136,A -71.3515,B 24.9635,C -1.3964,E1 25.0601,E2 517.7088} C_DIS
LIN {X 43.5968,Y -117.4307,Z 136,A -73.3609,B 24.9642,C -1.3828,E1 25.0548,E2 519.746} C_DIS
LIN {X 39.7543,Y -118.7861,Z 136,A -75.5615,B 24.9652,C -1.3638,E1 25.0488,E2 521.9873} C_DIS
LIN {X 36.221,Y -119.9115,Z 136,A -76.8827,B 24.9643,C -1.3803,E1 25.0454,E2 523.2672} C_DIS
LIN {X 32.4562,Y -120.9841,Z 136,A -78.687,B 24.9645,C -1.3776,E1 25.0405,E2 525.0748} C_DIS
LIN {X 28.5977,Y -121.9559,Z 136,A -80.4026,B 24.9643,C -1.3809,E1 25.0359,E2 526.7801} C_DIS
LIN {X 25.4072,Y -122.659,Z 136,A -82.3923,B 24.9656,C -1.3553,E1 25.0303,E2 528.828} C_DIS
LIN {X 21.5853,Y -123.3891,Z 136,A -83.8175,B 24.9648,C -1.3712,E1 25.0265,E2 530.214} C_DIS
LIN {X 17.7396,Y -123.9995,Z 136,A -85.5124,B 24.9646,C -1.3741,E1 25.0219,E2 531.9003} C_DIS
LIN {X 13.6799,Y -124.5132,Z 136,A -87.3756,B 24.9646,C -1.3734,E1 25.0167,E2 533.7639} C_DIS
LIN {X 10.3248,Y -124.8361,Z 136,A -88.9051,B 24.9646,C -1.3732,E1 25.0124,E2 535.293} C_DIS
LIN {X 6.4203,Y -125.0976,Z 136,A -90.7,B 24.9647,C -1.3722,E1 25.0074,E2 537.0896} C_DIS
LIN {X 2.6635,Y -125.2352,Z 136,A -92.5098,B 24.965,C -1.3672,E1 25.0024,E2 538.9108} C_DIS
LIN {X 2.6635,Y -125.2352,Z 136,A -92.5098,B 24.965,C -1.3672,E1 25.0024,E2 538.9108} C_DIS
Enddeposition()
LIN {X 0.8741,Y -124.2669,Z 136,A -92.7959,B 24.9627,C -1.4103,E1 25.0018,E2 539.0948} C_DIS
Startdeposition()
$VEL.CP = VEL_PRINT
LIN {X 3.9552,Y -124.2106,Z 136,A -91.0458,B 24.9619,C -1.4267,E1 25.0068,E2 537.3061} C_DIS
LIN {X 8.0004,Y -124.0153,Z 136,A -89.2021,B 24.9619,C -1.4263,E1 25.012,E2 535.4639} C_DIS
LIN {X 11.8961,Y -123.7018,Z 136,A -87.4418,B 24.9619,C -1.4253,E1 25.0169,E2 533.7072} C_DIS
LIN {X 16.0439,Y -123.2325,Z 136,A -85.5588,B 24.9619,C -1.4244,E1 25.0221,E2 531.8277} C_DIS
LIN {X 19.4811,Y -122.7369,Z 136,A -83.9233,B 24.9619,C -1.4273,E1 25.0266,E2 530.1869} C_DIS
LIN {X 24.1427,Y -121.9055,Z 136,A -81.5884,B 24.9613,C -1.4366,E1 25.0331,E2 527.8326} C_DIS
LIN {X 29.4841,Y -120.7246,Z 136,A -79.3187,B 24.9619,C -1.4265,E1 25.0392,E2 525.5899} C_DIS
LIN {X 32.9715,Y -119.8196,Z 136,A -76.55,B 24.9588,C -1.4839,E1 25.047,E2 522.69} C_DIS
LIN {X 39.4833,Y -117.8333,Z 136,A -74.5687,B 24.9617,C -1.4295,E1 25.0519,E2 520.8411} C_DIS
LIN {X 42.4224,Y -116.8075,Z 136,A -73.0363,B 24.9614,C -1.4362,E1 25.0559,E2 519.2959} C_DIS
LIN {X 46.5229,Y -115.2353,Z 136,A -70.6632,B 24.9603,C -1.4566,E1 25.0622,E2 516.8799} C_DIS
LIN {X 49.7883,Y -113.8637,Z 136,A -69.4628,B 24.9613,C -1.4373,E1 25.0652,E2 515.728} C_DIS
LIN {X 52.4103,Y -112.68,Z 136,A -68.0432,B 24.9609,C -1.4441,E1 25.0688,E2 514.2959} C_DIS
LIN {X 57.8482,Y -109.9869,Z 136,A -65.2421,B 24.9607,C -1.449,E1 25.0758,E2 511.4909} C_DIS
LIN {X 60.4756,Y -108.567,Z 136,A -63.8063,B 24.9604,C -1.4544,E1 25.0793,E2 510.0466} C_DIS
LIN {X 64.2364,Y -106.3847,Z 136,A -61.5743,B 24.9595,C -1.4697,E1 25.0847,E2 507.7853} C_DIS
LIN {X 67.1145,Y -104.5928,Z 136,A -60.4297,B 24.9605,C -1.4515,E1 25.0873,E2 506.6874} C_DIS
LIN {X 70.0712,Y -102.6359,Z 136,A -58.26,B 24.9589,C -1.482,E1 25.0925,E2 504.4528} C_DIS
LIN {X 73.3506,Y -100.3183,Z 136,A -56.9536,B 24.9602,C -1.4581,E1 25.0953,E2 503.2075} C_DIS
LIN {X 76.1506,Y -98.2094,Z 136,A -54.9069,B 24.9588,C -1.4836,E1 25.1,E2 501.108} C_DIS
LIN {X 78.9499,Y -95.9743,Z 136,A -53.1661,B 24.9583,C -1.4919,E1 25.1037,E2 499.3543} C_DIS
LIN {X 81.9714,Y -93.4059,Z 136,A -51.7913,B 24.9594,C -1.473,E1 25.1065,E2 498.0296} C_DIS
LIN {X 84.6784,Y -90.9591,Z 136,A -49.5664,B 24.9576,C -1.5049,E1 25.1112,E2 495.7385} C_DIS
LIN {X 87.9511,Y -87.7992,Z 136,A -47.5377,B 24.9575,C -1.5065,E1 25.1152,E2 493.7145} C_DIS
LIN {X 90.8878,Y -84.7551,Z 136,A -46.0616,B 24.9586,C -1.4871,E1 25.1179,E2 492.2907} C_DIS
LIN {X 93.7195,Y -81.6129,Z 136,A -43.5295,B 24.9566,C -1.5222,E1 25.1227,E2 489.6871} C_DIS
LIN {X 96.8525,Y -77.8693,Z 136,A -41.8682,B 24.958,C -1.4978,E1 25.1255,E2 488.0911} C_DIS
LIN {X 99.8778,Y -73.9496,Z 136,A -39.7283,B 24.958,C -1.4967,E1 25.1291,E2 485.964} C_DIS
LIN {X 102.7791,Y -69.8606,Z 136,A -37.3329,B 24.9574,C -1.5076,E1 25.133,E2 483.5547} C_DIS
LIN {X 105.7326,Y -65.3051,Z 136,A -34.7602,B 24.9568,C -1.5184,E1 25.1369,E2 480.9694} C_DIS
LIN {X 108.074,Y -61.3521,Z 136,A -32.6828,B 24.9566,C -1.5225,E1 25.1398,E2 478.8929} C_DIS
LIN {X 112.5559,Y -52.6787,Z 136,A -27.2025,B 24.9528,C -1.5873,E1 25.1467,E2 473.2892} C_DIS
LIN {X 115.3663,Y -46.198,Z 136,A -25.1587,B 24.9559,C -1.5341,E1 25.1487,E2 471.3821} C_DIS
LIN {X 116.4396,Y -43.4215,Z 136,A -23.7061,B 24.9554,C -1.5426,E1 25.1502,E2 469.9177} C_DIS
LIN {X 117.862,Y -39.3972,Z 136,A -21.0731,B 24.953,C -1.5835,E1 25.1526,E2 467.2031} C_DIS
LIN {X 119.3658,Y -34.5761,Z 136,A -19.4034,B 24.9546,C -1.5566,E1 25.1539,E2 465.6063} C_DIS
LIN {X 120.2431,Y -31.3944,Z 136,A -17.4013,B 24.9528,C -1.5865,E1 25.1553,E2 463.5452} C_DIS
LIN {X 121.2397,Y -27.2893,Z 136,A -15.9958,B 24.9541,C -1.5646,E1 25.1562,E2 462.1995} C_DIS
LIN {X 122.0086,Y -23.6136,Z 136,A -14.2542,B 24.9538,C -1.5708,E1 25.1571,E2 460.4535} C_DIS
LIN {X 122.5788,Y -20.4466,Z 136,A -12.7808,B 24.9535,C -1.5751,E1 25.1578,E2 458.9785} C_DIS
LIN {X 123.1521,Y -16.6572,Z 136,A -10.97,B 24.953,C -1.5832,E1 25.1585,E2 457.1594} C_DIS
LIN {X 123.5893,Y -13.0159,Z 136,A -9.2682,B 24.9527,C -1.5893,E1 25.1591,E2 455.4532} C_DIS
LIN {X 123.9449,Y -9.0179,Z 136,A -7.5138,B 24.9527,C -1.5904,E1 25.1594,E2 453.7066} C_DIS
LIN {X 124.1716,Y -5.0098,Z 136,A -5.6763,B 24.9523,C -1.5958,E1 25.1597,E2 451.8673} C_DIS
LIN {X 124.2651,Y -1.4829,Z 136,A -3.9645,B 24.9517,C -1.6056,E1 25.1597,E2 450.1427} C_DIS
LIN {X 124.2515,Y 2.3022,Z 136,A -2.2407,B 24.9514,C -1.6102,E1 25.1597,E2 448.4182} C_DIS
LIN {X 124.1049,Y 6.4565,Z 136,A -0.4816,B 24.9515,C -1.6083,E1 25.1595,E2 446.674} C_DIS
LIN {X 123.8619,Y 10.1,Z 136,A 1.2757,B 24.951,C -1.6176,E1 25.1591,E2 444.9052} C_DIS
LIN {X 123.4934,Y 13.907,Z 136,A 3.1558,B 24.9503,C -1.6294,E1 25.1586,E2 443.0086} C_DIS
LIN {X 123.0339,Y 17.5013,Z 136,A 4.6592,B 24.9504,C -1.6262,E1 25.158,E2 441.5216} C_DIS
LIN {X 122.5003,Y 20.9172,Z 136,A 6.5645,B 24.9491,C -1.6474,E1 25.1571,E2 439.5776} C_DIS
LIN {X 121.886,Y 24.2426,Z 136,A 8.6994,B 24.947,C -1.6824,E1 25.1559,E2 437.3726} C_DIS
LIN {X 120.5286,Y 30.2746,Z 136,A 10.3806,B 24.9502,C -1.6306,E1 25.1549,E2 435.823} C_DIS
LIN {X 117.8736,Y 39.3625,Z 136,A 14.9141,B 24.9488,C -1.6526,E1 25.1513,E2 431.2636} C_DIS
LIN {X 116.7669,Y 42.5349,Z 136,A 16.4415,B 24.9486,C -1.6562,E1 25.1498,E2 429.7364} C_DIS
LIN {X 115.7414,Y 45.2497,Z 136,A 17.7782,B 24.9484,C -1.6601,E1 25.1485,E2 428.3979} C_DIS
LIN {X 114.4897,Y 48.331,Z 136,A 19.3989,B 24.9478,C -1.6691,E1 25.1467,E2 426.7648} C_DIS
LIN {X 112.4426,Y 52.92,Z 136,A 21.7599,B 24.9472,C -1.6781,E1 25.144,E2 424.3954} C_DIS
LIN {X 110.5228,Y 56.8199,Z 136,A 23.6717,B 24.9472,C -1.6791,E1 25.1416,E2 422.4916} C_DIS
LIN {X 108.5503,Y 60.5058,Z 136,A 25.6613,B 24.9466,C -1.6876,E1 25.1389,E2 420.4923} C_DIS
LIN {X 106.3957,Y 64.2182,Z 136,A 27.5911,B 24.9464,C -1.6904,E1 25.1362,E2 418.5656} C_DIS
LIN {X 104.05,Y 67.9538,Z 136,A 29.6576,B 24.946,C -1.6975,E1 25.133,E2 416.4929} C_DIS
LIN {X 101.6222,Y 71.5328,Z 136,A 31.581,B 24.9459,C -1.6991,E1 25.13,E2 414.5751} C_DIS
LIN {X 99.1407,Y 74.9341,Z 136,A 33.5285,B 24.9456,C -1.7043,E1 25.1268,E2 412.6247} C_DIS
LIN {X 96.4614,Y 78.3539,Z 136,A 35.5667,B 24.9451,C -1.7109,E1 25.1232,E2 410.5804} C_DIS
LIN {X 93.6967,Y 81.6391,Z 136,A 37.5022,B 24.945,C -1.7134,E1 25.1197,E2 408.6479} C_DIS
LIN {X 89.8027,Y 85.9038,Z 136,A 39.9325,B 24.9453,C -1.7077,E1 25.1151,E2 406.2417} C_DIS
LIN {X 87.3873,Y 88.3603,Z 136,A 41.7381,B 24.9444,C -1.7221,E1 25.1115,E2 404.4097} C_DIS
LIN {X 84.3149,Y 91.2966,Z 136,A 43.699,B 24.9442,C -1.7263,E1 25.1075,E2 402.447} C_DIS
LIN {X 80.7953,Y 94.4261,Z 136,A 45.8409,B 24.944,C -1.7291,E1 25.103,E2 400.3067} C_DIS
LIN {X 77.5867,Y 97.0791,Z 136,A 48.1247,B 24.9425,C -1.7511,E1 25.098,E2 397.9797} C_DIS
LIN {X 74.4786,Y 99.4839,Z 136,A 49.5049,B 24.9437,C -1.7327,E1 25.095,E2 396.6478} C_DIS
LIN {X 71.3728,Y 101.7351,Z 136,A 51.3216,B 24.9434,C -1.7382,E1 25.0908,E2 394.8245} C_DIS
LIN {X 67.9293,Y 104.0658,Z 136,A 53.2621,B 24.9431,C -1.7426,E1 25.0863,E2 392.8802} C_DIS
LIN {X 64.2144,Y 106.398,Z 136,A 55.2502,B 24.943,C -1.744,E1 25.0816,E2 390.895} C_DIS
LIN {X 60.5332,Y 108.5352,Z 136,A 57.0739,B 24.9433,C -1.74,E1 25.0772,E2 389.0863} C_DIS
LIN {X 57.4719,Y 110.1846,Z 136,A 58.6754,B 24.9431,C -1.7421,E1 25.0732,E2 387.4842} C_DIS
LIN {X 54.4634,Y 111.7032,Z 136,A 60.3869,B 24.9425,C -1.7518,E1 25.0689,E2 385.7543} C_DIS
LIN {X 50.8577,Y 113.389,Z 136,A 62.0722,B 24.9428,C -1.7467,E1 25.0647,E2 384.0855} C_DIS
LIN {X 47.836,Y 114.6965,Z 136,A 63.5924,B 24.9428,C -1.7484,E1 25.0608,E2 382.5647} C_DIS
LIN {X 44.6118,Y 115.9894,Z 136,A 65.34,B 24.9421,C -1.7572,E1 25.0562,E2 380.8002} C_DIS
LIN {X 40.8768,Y 117.3571,Z 136,A 67.0372,B 24.9425,C -1.7522,E1 25.0518,E2 379.1183} C_DIS
LIN {X 37.6143,Y 118.4432,Z 136,A 68.6449,B 24.9423,C -1.7546,E1 25.0475,E2 377.508} C_DIS
LIN {X 31.2798,Y 120.2734,Z 136,A 71.6246,B 24.9423,C -1.7537,E1 25.0395,E2 374.5353} C_DIS
LIN {X 25.2568,Y 121.6796,Z 136,A 74.6403,B 24.9417,C -1.7632,E1 25.0312,E2 371.5013} C_DIS
LIN {X 21.3642,Y 122.4233,Z 136,A 76.4677,B 24.9417,C -1.7639,E1 25.0262,E2 369.6743} C_DIS
LIN {X 17.3837,Y 123.0507,Z 136,A 78.1673,B 24.9422,C -1.7568,E1 25.0216,E2 367.9929} C_DIS
LIN {X 12.9319,Y 123.5983,Z 136,A 80.1596,B 24.9424,C -1.7536,E1 25.0161,E2 366.0099} C_DIS
LIN {X 9.7432,Y 123.8919,Z 136,A 81.8506,B 24.9417,C -1.7639,E1 25.0113,E2 364.2951} C_DIS
LIN {X 5.818,Y 124.137,Z 136,A 83.655,B 24.9417,C -1.7635,E1 25.0063,E2 362.4925} C_DIS
LIN {X 1.9972,Y 124.2566,Z 136,A 85.3049,B 24.9421,C -1.7579,E1 25.0017,E2 360.856} C_DIS
LIN {X -1.9368,Y 124.2576,Z 136,A 87.1162,B 24.9421,C -1.7574,E1 24.9966,E2 359.046} C_DIS
LIN {X -5.488,Y 124.153,Z 136,A 88.8781,B 24.9418,C -1.7627,E1 24.9917,E2 357.2712} C_DIS
LIN {X -9.1008,Y 123.9388,Z 136,A 90.4459,B 24.9421,C -1.7573,E1 24.9874,E2 355.7157} C_DIS
LIN {X -13.3284,Y 123.5556,Z 136,A 92.3996,B 24.9422,C -1.7561,E1 24.9819,E2 353.7636} C_DIS
LIN {X -18.348,Y 122.9123,Z 136,A 94.6554,B 24.9425,C -1.751,E1 24.9757,E2 351.5184} C_DIS
LIN {X -21.5526,Y 122.3896,Z 136,A 96.2537,B 24.9423,C -1.7546,E1 24.9713,E2 349.9098} C_DIS
LIN {X -27.5515,Y 121.1798,Z 136,A 98.941,B 24.9429,C -1.7459,E1 24.964,E2 347.24} C_DIS
LIN {X -30.44,Y 120.4866,Z 136,A 100.8475,B 24.9413,C -1.7697,E1 24.9587,E2 345.2744} C_DIS
LIN {X -34.1638,Y 119.4862,Z 136,A 102.1512,B 24.9429,C -1.7456,E1 24.9553,E2 344.0259} C_DIS
LIN {X -38.2963,Y 118.2253,Z 136,A 104.1438,B 24.943,C -1.7433,E1 24.95,E2 342.0352} C_DIS
LIN {X -42.1644,Y 116.9005,Z 136,A 106.0587,B 24.9431,C -1.7423,E1 24.945,E2 340.1189} C_DIS
LIN {X -45.3187,Y 115.7146,Z 136,A 107.7031,B 24.943,C -1.7444,E1 24.9406,E2 338.4661} C_DIS
LIN {X -48.6689,Y 114.3466,Z 136,A 109.7866,B 24.9419,C -1.7612,E1 24.9352,E2 336.3378} C_DIS
LIN {X -52.1798,Y 112.7866,Z 136,A 111.0916,B 24.9435,C -1.7369,E1 24.932,E2 335.0874} C_DIS
LIN {X -55.3087,Y 111.2862,Z 136,A 112.6937,B 24.9436,C -1.7344,E1 24.928,E2 333.4871} C_DIS
LIN {X -59.0164,Y 109.3669,Z 136,A 114.5884,B 24.9439,C -1.7297,E1 24.9233,E2 331.5983} C_DIS
LIN {X -61.6228,Y 107.9196,Z 136,A 116.101,B 24.9437,C -1.7336,E1 24.9196,E2 330.072} C_DIS
LIN {X -65.0571,Y 105.8848,Z 136,A 118.2201,B 24.9431,C -1.743,E1 24.9145,E2 327.9241} C_DIS
LIN {X -67.8904,Y 104.0903,Z 136,A 119.5804,B 24.9438,C -1.7314,E1 24.9113,E2 326.5868} C_DIS
LIN {X -71.553,Y 101.608,Z 136,A 121.2875,B 24.9451,C -1.7121,E1 24.9075,E2 324.9199} C_DIS
LIN {X -73.8727,Y 99.9348,Z 136,A 122.8967,B 24.9444,C -1.7226,E1 24.9038,E2 323.2802} C_DIS
Enddeposition()
END
